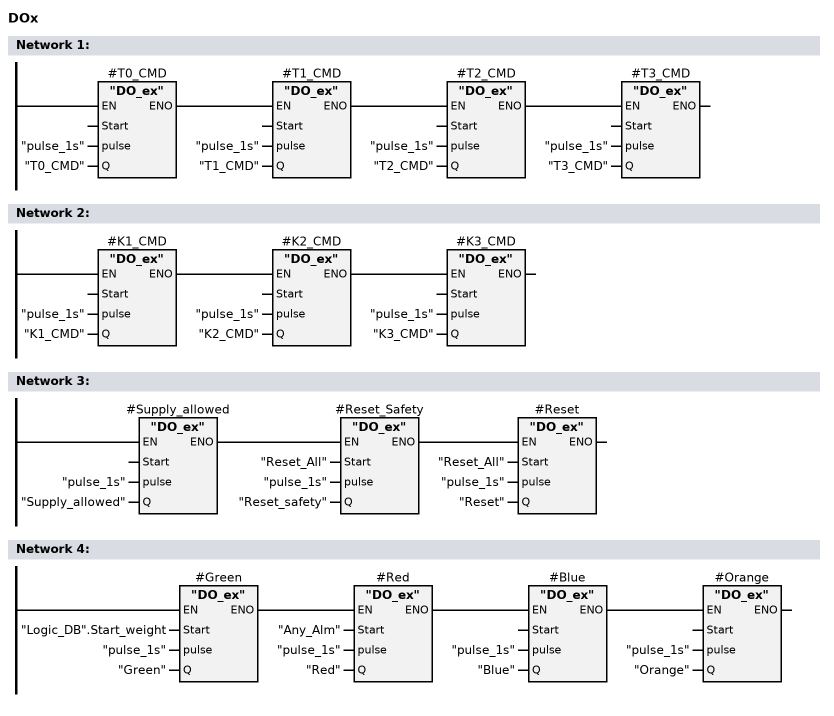
   RUNG wire#powerrail
      #T0_CMD(pulse := "pulse_1s", Q := "T0_CMD", Start :=)
      #T1_CMD(pulse := "pulse_1s", Q := "T1_CMD", Start :=)
      #T2_CMD(pulse := "pulse_1s", Q := "T2_CMD", Start :=)
      #T3_CMD(pulse := "pulse_1s", Q := "T3_CMD", Start :=)
   END_RUNG
   // the same network as SCL:
   #T0_CMD(pulse := "pulse_1s", Q := "T0_CMD", ENO => #_w1);   // "DO_ex"
   #T1_CMD(EN := #_w1, pulse := "pulse_1s", Q := "T1_CMD", ENO => #_w2);   // "DO_ex"
   #T2_CMD(EN := #_w2, pulse := "pulse_1s", Q := "T2_CMD", ENO => #_w3);   // "DO_ex"
   IF #_w3 THEN
       #T3_CMD(pulse := "pulse_1s", Q := "T3_CMD");   // "DO_ex"
   END_IF;
END_REGION

REGION Network 2
   RUNG wire#powerrail
      #K1_CMD(pulse := "pulse_1s", Q := "K1_CMD", Start :=)
      #K2_CMD(pulse := "pulse_1s", Q := "K2_CMD", Start :=)
      #K3_CMD(pulse := "pulse_1s", Q := "K3_CMD", Start :=)
   END_RUNG
   // the same network as SCL:
   #K1_CMD(pulse := "pulse_1s", Q := "K1_CMD", ENO => #_w1);   // "DO_ex"
   #K2_CMD(EN := #_w1, pulse := "pulse_1s", Q := "K2_CMD", ENO => #_w2);   // "DO_ex"
   IF #_w2 THEN
       #K3_CMD(pulse := "pulse_1s", Q := "K3_CMD");   // "DO_ex"
   END_IF;
END_REGION

REGION Network 3
   RUNG wire#powerrail
      #Supply_allowed(Start :=, pulse := "pulse_1s", Q := "Supply_allowed")
      #Reset_Safety(Start := "Reset_All", pulse := "pulse_1s", Q := "Reset_safety")
      #Reset(Start := "Reset_All", pulse := "pulse_1s", Q := "Reset")
   END_RUNG
   // the same network as SCL:
   #Supply_allowed(pulse := "pulse_1s", Q := "Supply_allowed", ENO => #_w1);   // "DO_ex"
   #Reset_Safety(EN := #_w1, Start := "Reset_All", pulse := "pulse_1s", Q := "Reset_safety", ENO => #_w2);   // "DO_ex"
   IF #_w2 THEN
       #Reset(Start := "Reset_All", pulse := "pulse_1s", Q := "Reset");   // "DO_ex"
   END_IF;
END_REGION

REGION Network 4
   RUNG wire#powerrail
      #Green(Start := "Logic_DB".Start_weight, pulse := "pulse_1s", Q := "Green")
      #Red(Start := "Any_Alm", pulse := "pulse_1s", Q := "Red")
      #Blue(Start :=, pulse := "pulse_1s", Q := "Blue")
      #Orange(Start :=, pulse := "pulse_1s", Q := "Orange")
   END_RUNG
   // the same network as SCL:
   #Green(Start := "Logic_DB".Start_weight, pulse := "pulse_1s", Q := "Green", ENO => #_w1);   // "DO_ex"
   #Red(EN := #_w1, Start := "Any_Alm", pulse := "pulse_1s", Q := "Red", ENO => #_w2);   // "DO_ex"
   #Blue(EN := #_w2, pulse := "pulse_1s", Q := "Blue", ENO => #_w3);   // "DO_ex"
   IF #_w3 THEN
       #Orange(pulse := "pulse_1s", Q := "Orange");   // "DO_ex"
   END_IF;
END_REGION
END_FUNCTION_BLOCK

// folder: System

FUNCTION_BLOCK "Tachometer"   // FB98, LAD
{ S7_Optimized_Access := 'FALSE' }
VERSION : 0.1
   VAR_INPUT
      Run : Bool;   // Управляющий сигнал
      Add : Bool;   // Один импульс
   END_VAR
   VAR_IN_OUT
      Result : Real;   // Текущая скорость, %
   END_VAR
   VAR
      Full : Real := 10.0;   // Кол-во импульсов на 1 оборот
      One : Real;   // Вес 1 импульса
      "A" : Real;   // Суммарный вес импульсов
      "B" : Real;   // Вес за последний цикл измерений
      T : Struct   // Уставка = времени одного оборота при 100% скорости
         SP : Real := 10.0;   // Уставка
         Now : Real;   // Текущий счёт
         One : Real;   // Вес импульса
         Progress : Real;   // Прогресс выполнения
         "Exit" : Bool;   // Счёт завершён
         Start : Bool;   // Запуск
         Pause : Bool;   // Пауза
         Reset : Bool;
         pos : Bool;   // Контроль фронта сигнала
      END_STRUCT;
   END_VAR
   VAR_TEMP
      pos_1 : Bool;
   END_VAR
   VAR_TEMP   // added for the SCL form of the ladder/FBD networks
      _w1 : Bool;
   END_VAR
BEGIN

REGION Network 1: Рассчёт веса импульса
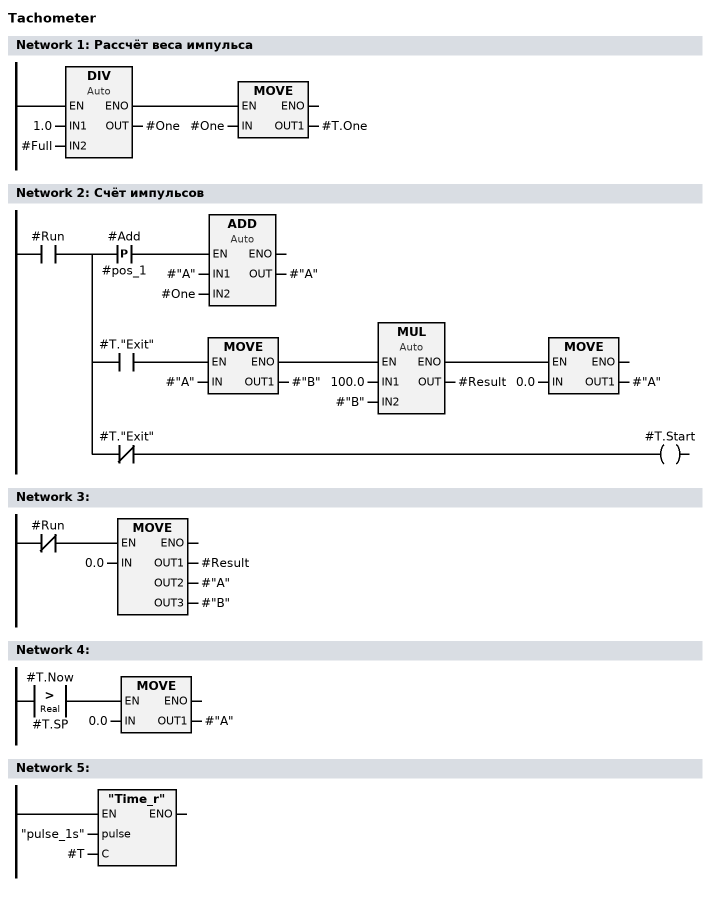
   RUNG wire#powerrail
      Div(in1 := 1.0, in2 := #Full, out => #One)
      Move(in := #One, out1 => #T.One)
   END_RUNG
   // the same network as SCL:
   #One := 1.0 / #Full;
   #T.One := #One;
END_REGION

REGION Network 2: Счёт импульсов
   RUNG wire#powerrail
      Contact( #Run )
      wire#w1
      P_Contact(operand := #Add, bit := #pos_1)
      Add(in1 := #"A", in2 := #One, out => #"A")
   END_RUNG
   RUNG wire#w1
      Contact( #T."Exit" )
      Move(in := #"A", out1 => #"B")
      Mul(in1 := 100.0, in2 := #"B", out => #Result)
      Move(in := 0.0, out1 => #"A")
   END_RUNG
   RUNG wire#w1
      I_Contact( #T."Exit" )
      Coil( #T.Start )
   END_RUNG
   // the same network as SCL:
   #_w1 := #Run AND #Add AND NOT #pos_1;   // rising edge of #Add
   #pos_1 := #Add;
   IF #_w1 THEN #"A" := #"A" + #One; END_IF;
   IF #Run AND #T."Exit" THEN
       #"B" := #"A";
       #Result := 100.0 * #"B";
       #"A" := 0.0;
   END_IF;
   #T.Start := #Run AND NOT #T."Exit";
END_REGION

REGION Network 3
   RUNG wire#powerrail
      I_Contact( #Run )
      Move(in := 0.0, out1 => #Result, out2 => #"A", out3 => #"B")
   END_RUNG
   // the same network as SCL:
   IF NOT #Run THEN
       #Result := 0.0;
       #"A" := 0.0;
       #"B" := 0.0;
   END_IF;
END_REGION

REGION Network 4
   RUNG wire#powerrail
      { S7_Templates := "SrcType := Real" } GT_Contact(in1 := #T.Now, in2 := #T.SP)
      Move(in := 0.0, out1 => #"A")
   END_RUNG
   // the same network as SCL:
   IF #T.Now > #T.SP THEN #"A" := 0.0; END_IF;
END_REGION

REGION Network 5
   RUNG wire#powerrail
      "Time_r"(pulse := "pulse_1s", C := #T)
   END_RUNG
   // the same network as SCL:
   "Time_r"(pulse := "pulse_1s", C := #T);
END_REGION
END_FUNCTION_BLOCK

FUNCTION_BLOCK "PID_ex"   // FB99, LAD
{ S7_Optimized_Access := 'FALSE' }
VERSION : 0.1
   VAR_INPUT
      Start : Bool;   // Команда запуска
      SP : Real;   // Уставка
      Value : Real;   // Показания датчика
   END_VAR
   VAR_IN_OUT
      Result : Real;   // Управляющее воздействие
   END_VAR
   VAR
      Hand : Bool;   // Ручной режим
      Err_Ack : Bool;   // Подтверждение аварии
      Reset : Bool;   // Сброс ПИД
      Error : Bool;   // Авария ПИД
      Invert : Bool;   // Инверсия работы
      SP_H : Bool;   // Авария уставки - превышение
      SP_L : Bool;   // Авария уставки - занижение
      In_H : Bool;   // Авария датчика - превышение
      In_L : Bool;   // Авария датчика - занижение
      Activate : Bool;   // Активировать ПИД
      Error_code : DWord;   // Код аварии
      Warning_code : DWord;   // Код предупреждения
      HandValue : Real;   // Выход ПИД в ручном режиме
      SP_P : Real := 1.5;   // Коэффициент пропорциональности
      SP_Ti : Real := 150.0;   // Время интегрирования
      SP_Td : Real;   // Время дифференцирования
      SP_Cycle : Real := 0.2;   // Время цикла
      Disturvance : Real;   // Внешнее воздействие
      Max_SP : Real := 500.0;   // Максимальное значение уставки
      Min_SP : Real := -500.0;   // Минимальное значение уставки
      Max_in : Real := 500.0;   // Максимальное значение датчика
      Min_in : Real := -500.0;   // Минимальное значение датчика
      Max_out : Real := 100.0;   // Максимальное значение выхода
      Min_out : Real := 0.0;   // Минимальное значение выхода
      "Type" : Int := 1;   // Режим работы
      State : Int;   // Состояние
      Mode : Int := 3;   // Режим
      PID : PID_Compact;   // ПИД
      DeadBand : Real;   // Мёртвая зона
      Max : Real;   // Верняя граница мёртвой зоны
      Min : Real;   // Нижняя граница мёртвой зоны
      Converter : Struct
         Use_Min_In : Bool;   // Отсекать входные значения ниже минимума
         Use_Max_In : Bool;   // Отсекать входные значения выше максимума
         Use_Min_Out : Bool;   // Отсекать результат ниже минимума
         Use_Max_Out : Bool;   // Отсекать результат выше максимума
         IO : Bool;   // Входной/Выходной режим
         Inverse : Bool;   // Инверсия выхода
         Min_In : Real := 0.0;   // Минимальный входной сигнал
         Max_In : Real := 100.0;   // Максимальный входной сигнал
         Min_Out : Real;   // Минимальный выходной сигнал
         Max_Out : Real;   // Максимальный выходной сигнал
      END_STRUCT;
      Conveter_Back : Struct
         Use_Min_In : Bool;   // Отсекать входные значения ниже минимума
         Use_Max_In : Bool;   // Отсекать входные значения выше максимума
         Use_Min_Out : Bool;   // Отсекать результат ниже минимума
         Use_Max_Out : Bool;   // Отсекать результат выше максимума
         IO : Bool;   // Входной/Выходной режим
         Inverse : Bool;   // Инверсия выхода
         Min_In : Real;   // Минимальный входной сигнал
         Max_In : Real;   // Максимальный входной сигнал
         Min_Out : Real := 0.0;   // Минимальный выходной сигнал
         Max_Out : Real := 100.0;   // Максимальный выходной сигнал
      END_STRUCT;
      C : Struct
         SP : Real := 1.0;   // Уставка
         Now : Real;   // Текущий счёт
         One : Real;   // Вес импульса
         Progress : Real;   // Прогресс выполнения
         "Exit" : Bool;   // Счёт завершён
         Start : Bool;   // Запуск
         Pause : Bool;   // Пауза
         Reset : Bool;   // Сброс счёта
         pos : Bool;   // Контроль фронта сигнала
      END_STRUCT;
   END_VAR
   VAR_TEMP
      PID_Output : Real;
   END_VAR
   VAR_TEMP   // added for the SCL form of the ladder/FBD networks
      _w1 : Bool;
   END_VAR
BEGIN

REGION Network 1: Сброс ПИД
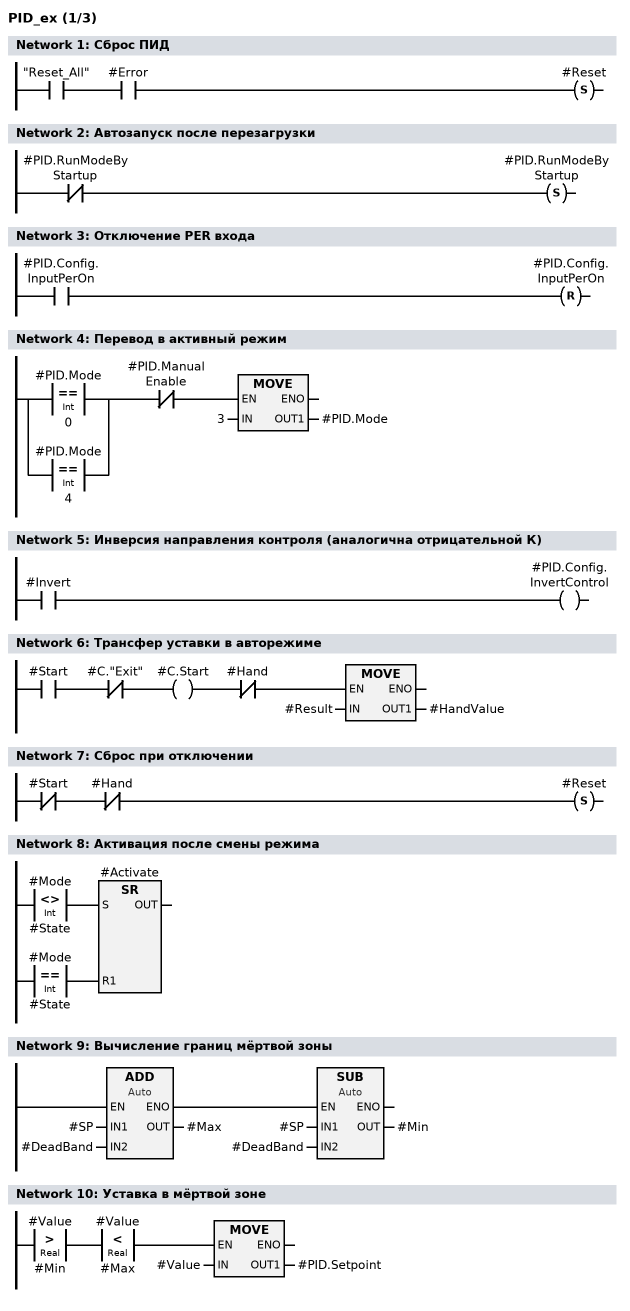
   RUNG wire#powerrail
      Contact( "Reset_All" )
      Contact( #Error )
      S_Coil( #Reset )
   END_RUNG
   // the same network as SCL:
   IF "Reset_All" AND #Error THEN #Reset := TRUE; END_IF;
END_REGION

REGION Network 2: Автозапуск после перезагрузки
   RUNG wire#powerrail
      I_Contact( #PID.RunModeByStartup )
      S_Coil( #PID.RunModeByStartup )
   END_RUNG
   // the same network as SCL:
   IF NOT #PID.RunModeByStartup THEN #PID.RunModeByStartup := TRUE; END_IF;
END_REGION

REGION Network 3: Отключение PER входа
   RUNG wire#powerrail
      Contact( #PID.Config.InputPerOn )
      R_Coil( #PID.Config.InputPerOn )
   END_RUNG
   // the same network as SCL:
   IF #PID.Config.InputPerOn THEN #PID.Config.InputPerOn := FALSE; END_IF;
END_REGION

REGION Network 4: Перевод в активный режим
   RUNG wire#powerrail
      { S7_Templates := "SrcType := Int" } EQ_Contact(in1 := #PID.Mode, in2 := 0)
      wire#w1
      I_Contact( #PID.ManualEnable )
      { S7_GenerateENO := "TRUE" } Move(in := 3, out1 => #PID.Mode)
   END_RUNG
   RUNG wire#powerrail
      { S7_Templates := "SrcType := Int" } EQ_Contact(in1 := #PID.Mode, in2 := 4)
   END_RUNG wire#w1
   // the same network as SCL:
   IF ((#PID.Mode = 0) OR (#PID.Mode = 4)) AND NOT #PID.ManualEnable THEN #PID.Mode := 3; END_IF;
END_REGION

REGION Network 5: Инверсия направления контроля (аналогична отрицательной К)
   RUNG wire#powerrail
      Contact( #Invert )
      Coil( #PID.Config.InvertControl )
   END_RUNG
   // the same network as SCL:
   #PID.Config.InvertControl := #Invert;
END_REGION

REGION Network 6: Трансфер уставки в авторежиме
   RUNG wire#powerrail
      Contact( #Start )
      I_Contact( #C."Exit" )
      Coil( #C.Start )
      I_Contact( #Hand )
      Move(in := #Result, out1 => #HandValue)
   END_RUNG
   // the same network as SCL:
   #C.Start := #Start AND NOT #C."Exit";
   IF #C.Start AND NOT #Hand THEN #HandValue := #Result; END_IF;
END_REGION

REGION Network 7: Сброс при отключении
   RUNG wire#powerrail
      I_Contact( #Start )
      I_Contact( #Hand )
      S_Coil( #Reset )
   END_RUNG
   // the same network as SCL:
   IF NOT #Start AND NOT #Hand THEN #Reset := TRUE; END_IF;
END_REGION

REGION Network 8: Активация после смены режима
   RUNG wire#powerrail
      { S7_Templates := "SrcType := Int" } NE_Contact(in1 := #Mode, in2 := #State)
      S_SR(operand := #Activate, r1 := wire#w1)
   END_RUNG
   RUNG wire#powerrail
      { S7_Templates := "SrcType := Int" } EQ_Contact(in1 := #Mode, in2 := #State)
   END_RUNG wire#w1
   // the same network as SCL:
   IF #Mode <> #State THEN
       #Activate := TRUE;   // SR flip-flop
   END_IF;
   IF #Mode = #State THEN #Activate := FALSE; END_IF;
END_REGION

REGION Network 9: Вычисление границ мёртвой зоны
   RUNG wire#powerrail
      Add(in1 := #SP, in2 := #DeadBand, out => #Max)
      Sub(in1 := #SP, in2 := #DeadBand, out => #Min)
   END_RUNG
   // the same network as SCL:
   #Max := #SP + #DeadBand;
   #Min := #SP - #DeadBand;
END_REGION

REGION Network 10: Уставка в мёртвой зоне
   RUNG wire#powerrail
      { S7_Templates := "SrcType := Real" } GT_Contact(in1 := #Value, in2 := #Min)
      { S7_Templates := "SrcType := Real" } LT_Contact(in1 := #Value, in2 := #Max)
      Move(in := #Value, out1 => #PID.Setpoint)
   END_RUNG
   // the same network as SCL:
   IF (#Value > #Min) AND (#Value < #Max) THEN #PID.Setpoint := #Value; END_IF;
END_REGION

REGION Network 11: Уставка вне мёртвой зоны
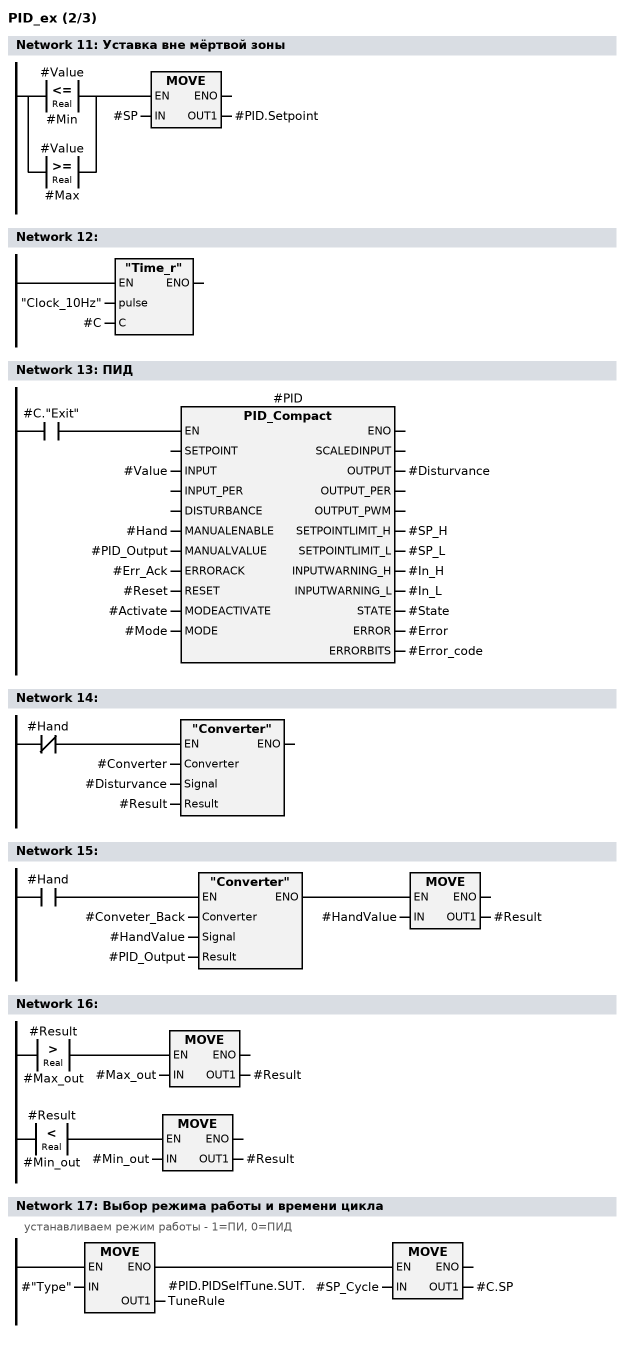
   RUNG wire#powerrail
      { S7_Templates := "SrcType := Real" } LE_Contact(in1 := #Value, in2 := #Min)
      wire#w1
      Move(in := #SP, out1 => #PID.Setpoint)
   END_RUNG
   RUNG wire#powerrail
      { S7_Templates := "SrcType := Real" } GE_Contact(in1 := #Value, in2 := #Max)
   END_RUNG wire#w1
   // the same network as SCL:
   IF (#Value <= #Min) OR (#Value >= #Max) THEN #PID.Setpoint := #SP; END_IF;
END_REGION

REGION Network 12
   RUNG wire#powerrail
      "Time_r"(pulse := "Clock_10Hz", C := #C)
   END_RUNG
   // the same network as SCL:
   "Time_r"(pulse := "Clock_10Hz", C := #C);
END_REGION

REGION Network 13: ПИД
   IF #C."Exit" THEN
       #PID(Input := #Value,   // PID_Compact
            ManualEnable := #Hand,
            ManualValue := #PID_Output,
            ErrorAck := #Err_Ack,
            Reset := #Reset,
            ModeActivate := #Activate,
            Mode := #Mode,
            Output => #Disturvance,
            SetpointLimit_H => #SP_H,
            SetpointLimit_L => #SP_L,
            InputWarning_H => #In_H,
            InputWarning_L => #In_L,
            State => #State,
            Error => #Error,
            ErrorBits => #Error_code);
   END_IF;
END_REGION

REGION Network 14
   RUNG wire#powerrail
      I_Contact( #Hand )
      "Converter"(Converter := #Converter, Signal := #Disturvance, Result := #Result)
   END_RUNG
   // the same network as SCL:
   IF NOT #Hand THEN "Converter"(Converter := #Converter, Signal := #Disturvance, Result := #Result); END_IF;
END_REGION

REGION Network 15
   RUNG wire#powerrail
      Contact( #Hand )
      "Converter"(Converter := #Conveter_Back, Signal := #HandValue, Result := #PID_Output)
      Move(in := #HandValue, out1 => #Result)
   END_RUNG
   // the same network as SCL:
   "Converter"(EN := #Hand,
               Converter := #Conveter_Back,
               Signal := #HandValue,
               Result := #PID_Output,
               ENO => #_w1);
   IF #_w1 THEN #Result := #HandValue; END_IF;
END_REGION

REGION Network 16
   RUNG wire#powerrail
      { S7_Templates := "SrcType := Real" } GT_Contact(in1 := #Result, in2 := #Max_out)
      Move(in := #Max_out, out1 => #Result)
   END_RUNG
   RUNG wire#powerrail
      { S7_Templates := "SrcType := Real" } LT_Contact(in1 := #Result, in2 := #Min_out)
      Move(in := #Min_out, out1 => #Result)
   END_RUNG
   // the same network as SCL:
   IF #Result > #Max_out THEN #Result := #Max_out; END_IF;
   IF #Result < #Min_out THEN #Result := #Min_out; END_IF;
END_REGION

REGION Network 17: Выбор режима работы и времени цикла
   // устанавливаем режим работы - 1=ПИ, 0=ПИД
   RUNG wire#powerrail
      { S7_GenerateENO := "TRUE" } Move(in := #"Type", out1 => #PID.PIDSelfTune.SUT.TuneRule)
      { S7_GenerateENO := "TRUE" } Move(in := #SP_Cycle, out1 => #C.SP)
   END_RUNG
   // the same network as SCL:
   // ENO of a box is taken as its EN; it also drops when the box reports an error
   #PID.PIDSelfTune.SUT.TuneRule := #"Type";
   #C.SP := #SP_Cycle;
END_REGION

REGION Network 18: Параметры регулирования
   // Задаём коэффициент пропорциональности и время интегрирования.
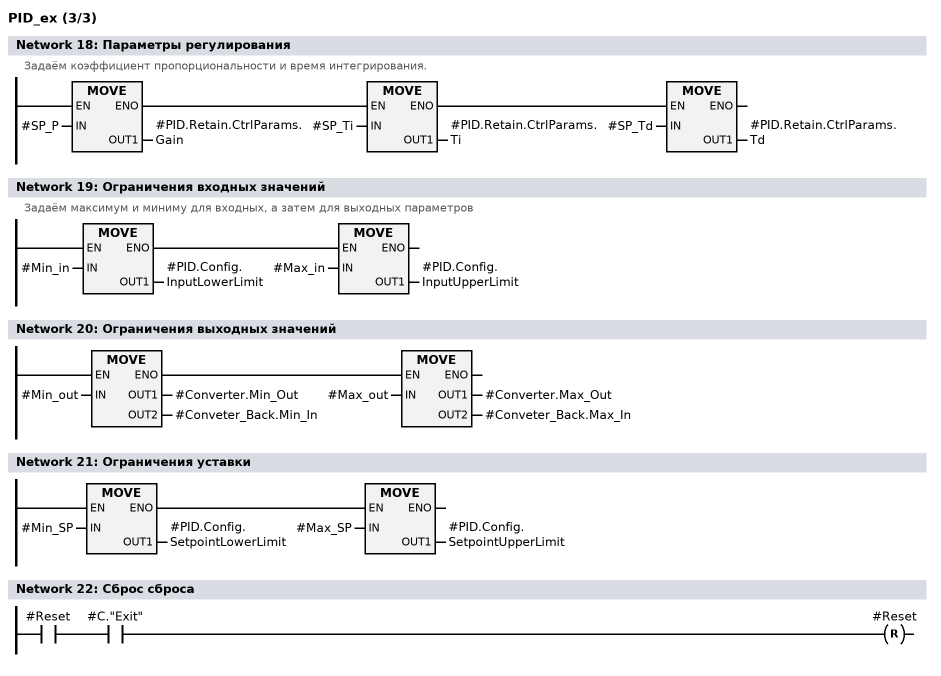
   RUNG wire#powerrail
      { S7_GenerateENO := "TRUE" } Move(in := #SP_P, out1 => #PID.Retain.CtrlParams.Gain)
      { S7_GenerateENO := "TRUE" } Move(in := #SP_Ti, out1 => #PID.Retain.CtrlParams.Ti)
      { S7_GenerateENO := "TRUE" } Move(in := #SP_Td, out1 => #PID.Retain.CtrlParams.Td)
   END_RUNG
   // the same network as SCL:
   // ENO of a box is taken as its EN; it also drops when the box reports an error
   #PID.Retain.CtrlParams.Gain := #SP_P;
   #PID.Retain.CtrlParams.Ti := #SP_Ti;
   #PID.Retain.CtrlParams.Td := #SP_Td;
END_REGION

REGION Network 19: Ограничения входных значений
   // Задаём максимум и миниму для входных, а затем для выходных параметров
   RUNG wire#powerrail
      { S7_GenerateENO := "TRUE" } Move(in := #Min_in, out1 => #PID.Config.InputLowerLimit)
      { S7_GenerateENO := "TRUE" } Move(in := #Max_in, out1 => #PID.Config.InputUpperLimit)
   END_RUNG
   // the same network as SCL:
   // ENO of a box is taken as its EN; it also drops when the box reports an error
   #PID.Config.InputLowerLimit := #Min_in;
   #PID.Config.InputUpperLimit := #Max_in;
END_REGION

REGION Network 20: Ограничения выходных значений
   RUNG wire#powerrail
      { S7_GenerateENO := "TRUE" } Move(in := #Min_out, out1 => #Converter.Min_Out, out2 => #Conveter_Back.Min_In)
      { S7_GenerateENO := "TRUE" } Move(in := #Max_out, out1 => #Converter.Max_Out, out2 => #Conveter_Back.Max_In)
   END_RUNG
   // the same network as SCL:
   // ENO of a box is taken as its EN; it also drops when the box reports an error
   #Converter.Min_Out := #Min_out;
   #Conveter_Back.Min_In := #Min_out;
   #Converter.Max_Out := #Max_out;
   #Conveter_Back.Max_In := #Max_out;
END_REGION

REGION Network 21: Ограничения уставки
   RUNG wire#powerrail
      { S7_GenerateENO := "TRUE" } Move(in := #Min_SP, out1 => #PID.Config.SetpointLowerLimit)
      { S7_GenerateENO := "TRUE" } Move(in := #Max_SP, out1 => #PID.Config.SetpointUpperLimit)
   END_RUNG
   // the same network as SCL:
   // ENO of a box is taken as its EN; it also drops when the box reports an error
   #PID.Config.SetpointLowerLimit := #Min_SP;
   #PID.Config.SetpointUpperLimit := #Max_SP;
END_REGION

REGION Network 22: Сброс сброса
   RUNG wire#powerrail
      Contact( #Reset )
      Contact( #C."Exit" )
      R_Coil( #Reset )
   END_RUNG
   // the same network as SCL:
   IF #Reset AND #C."Exit" THEN #Reset := FALSE; END_IF;
END_REGION
END_FUNCTION_BLOCK

FUNCTION "DRV_pulse" : Void   // FC100, LAD
{ S7_Optimized_Access := 'FALSE' }
VERSION : 0.1
   VAR_TEMP   // added for the SCL form of the ladder/FBD networks
      _w1 : Bool;
      _w2 : Bool;
   END_VAR
BEGIN

REGION Network 1
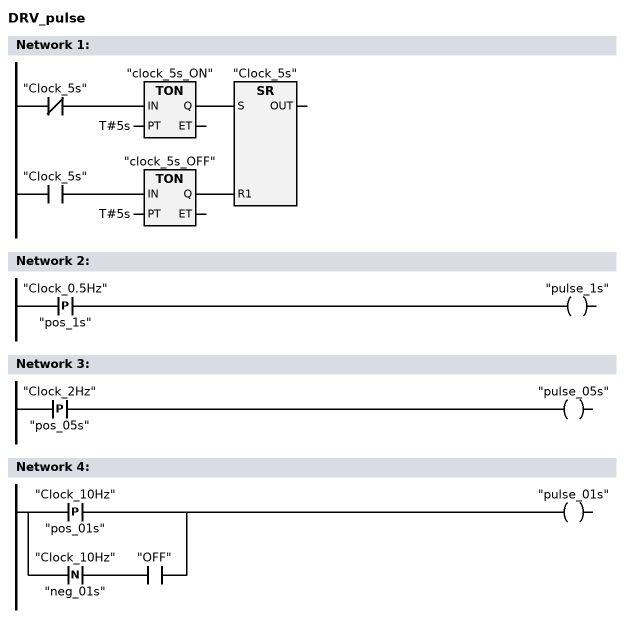
   "clock_5s_ON".TON(IN := NOT "Clock_5s", PT := T#5s);
   "clock_5s_OFF".TON(IN := "Clock_5s", PT := T#5s);
   IF "clock_5s_ON".Q THEN
       "Clock_5s" := TRUE;   // SR flip-flop
   END_IF;
   IF "clock_5s_OFF".Q THEN "Clock_5s" := FALSE; END_IF;
END_REGION

REGION Network 2
   RUNG wire#powerrail
      P_Contact(operand := "Clock_0.5Hz", bit := "pos_1s")
      Coil( "pulse_1s" )
   END_RUNG
   // the same network as SCL:
   #_w1 := "Clock_0.5Hz" AND NOT "pos_1s";   // rising edge of "Clock_0.5Hz"
   "pos_1s" := "Clock_0.5Hz";
   "pulse_1s" := #_w1;
END_REGION

REGION Network 3
   RUNG wire#powerrail
      P_Contact(operand := "Clock_2Hz", bit := "pos_05s")
      Coil( "pulse_05s" )
   END_RUNG
   // the same network as SCL:
   #_w1 := "Clock_2Hz" AND NOT "pos_05s";   // rising edge of "Clock_2Hz"
   "pos_05s" := "Clock_2Hz";
   "pulse_05s" := #_w1;
END_REGION

REGION Network 4
   RUNG wire#powerrail
      P_Contact(operand := "Clock_10Hz", bit := "pos_01s")
      wire#w1
      Coil( "pulse_01s" )
   END_RUNG
   RUNG wire#powerrail
      N_Contact(operand := "Clock_10Hz", bit := "neg_01s")
      Contact( "OFF" )
   END_RUNG wire#w1
   // the same network as SCL:
   #_w1 := "Clock_10Hz" AND NOT "pos_01s";   // rising edge of "Clock_10Hz"
   "pos_01s" := "Clock_10Hz";
   #_w2 := NOT "Clock_10Hz" AND "neg_01s";   // falling edge of "Clock_10Hz"
   "neg_01s" := "Clock_10Hz";
   "pulse_01s" := #_w1 OR (#_w2 AND "OFF");
END_REGION
END_FUNCTION

FUNCTION "DRV_End" : Void   // FC101, LAD
{ S7_Optimized_Access := 'TRUE' }
VERSION : 0.1
BEGIN

REGION Network 1: Одно из устройств нижнего уровня в ручном режиме
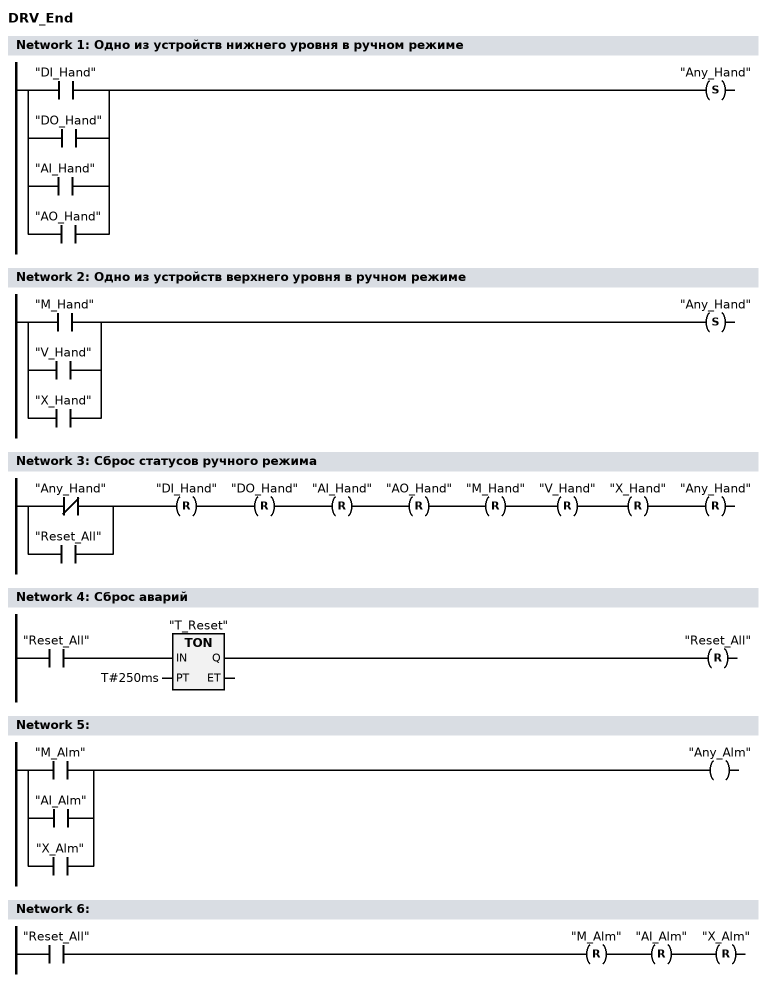
   RUNG wire#powerrail
      Contact( "DI_Hand" )
      wire#w1
      S_Coil( "Any_Hand" )
   END_RUNG
   RUNG wire#powerrail
      Contact( "DO_Hand" )
   END_RUNG wire#w1
   RUNG wire#powerrail
      Contact( "AI_Hand" )
   END_RUNG wire#w1
   RUNG wire#powerrail
      Contact( "AO_Hand" )
   END_RUNG wire#w1
   // the same network as SCL:
   IF "DI_Hand" OR "DO_Hand" OR "AI_Hand" OR "AO_Hand" THEN "Any_Hand" := TRUE; END_IF;
END_REGION

REGION Network 2: Одно из устройств верхнего уровня в ручном режиме
   RUNG wire#powerrail
      Contact( "M_Hand" )
      wire#w1
      S_Coil( "Any_Hand" )
   END_RUNG
   RUNG wire#powerrail
      Contact( "V_Hand" )
   END_RUNG wire#w1
   RUNG wire#powerrail
      Contact( "X_Hand" )
   END_RUNG wire#w1
   // the same network as SCL:
   IF "M_Hand" OR "V_Hand" OR "X_Hand" THEN "Any_Hand" := TRUE; END_IF;
END_REGION

REGION Network 3: Сброс статусов ручного режима
   RUNG wire#powerrail
      I_Contact( "Any_Hand" )
      wire#w1
      R_Coil( "DI_Hand" )
      R_Coil( "DO_Hand" )
      R_Coil( "AI_Hand" )
      R_Coil( "AO_Hand" )
      R_Coil( "M_Hand" )
      R_Coil( "V_Hand" )
      R_Coil( "X_Hand" )
      R_Coil( "Any_Hand" )
   END_RUNG
   RUNG wire#powerrail
      Contact( "Reset_All" )
   END_RUNG wire#w1
   // the same network as SCL:
   IF NOT "Any_Hand" OR "Reset_All" THEN
       "DI_Hand" := FALSE;
       "DO_Hand" := FALSE;
       "AI_Hand" := FALSE;
       "AO_Hand" := FALSE;
       "M_Hand" := FALSE;
       "V_Hand" := FALSE;
       "X_Hand" := FALSE;
       "Any_Hand" := FALSE;
   END_IF;
END_REGION

REGION Network 4: Сброс аварий
   "T_Reset".TON(IN := "Reset_All", PT := T#250ms);
   IF "T_Reset".Q THEN "Reset_All" := FALSE; END_IF;
END_REGION

REGION Network 5
   RUNG wire#powerrail
      Contact( "M_Alm" )
      wire#w1
      Coil( "Any_Alm" )
   END_RUNG
   RUNG wire#powerrail
      Contact( "AI_Alm" )
   END_RUNG wire#w1
   RUNG wire#powerrail
      Contact( "X_Alm" )
   END_RUNG wire#w1
   // the same network as SCL:
   "Any_Alm" := "M_Alm" OR "AI_Alm" OR "X_Alm";
END_REGION

REGION Network 6
   RUNG wire#powerrail
      Contact( "Reset_All" )
      R_Coil( "M_Alm" )
      R_Coil( "AI_Alm" )
      R_Coil( "X_Alm" )
   END_RUNG
   // the same network as SCL:
   IF "Reset_All" THEN
       "M_Alm" := FALSE;
       "AI_Alm" := FALSE;
       "X_Alm" := FALSE;
   END_IF;
END_REGION
END_FUNCTION

FUNCTION "Converter" : Void   // FC102, LAD
TITLE = Драйвер линеаризации аналогового сигнала
{ S7_Optimized_Access := 'FALSE' }
VERSION : 0.1
   VAR_INPUT
      Converter : Struct
         Use_Min_In : Bool;   // Отсекать входные значения ниже минимума
         Use_Max_In : Bool;   // Отсекать входные значения выше максимума
         Use_Min_Out : Bool;   // Отсекать результат ниже минимума
         Use_Max_Out : Bool;   // Отсекать результат выше максимума
         IO : Bool;   // Входной/Выходной режим
         Inverse : Bool;   // Инверсия выхода
         Min_In : Real;   // Минимальный входной сигнал
         Max_In : Real;   // Максимальный входной сигнал
         Min_Out : Real;   // Минимальный выходной сигнал
         Max_Out : Real;   // Максимальный выходной сигнал
      END_STRUCT;
   END_VAR
   VAR_IN_OUT
      Signal : Real;   // Входной сигнал
      Result : Real;   // Результат линеаризации
   END_VAR
   VAR_TEMP
      Range_In : Real;   // Диапазон входного сигнала
      Range_Out : Real;   // Диапазон выходного сигнала
      T_T : Real;   // Соотношение диапазонов
      R_Sig : Real;   // Поправка на отрицательные значения
   END_VAR
BEGIN

REGION Network 1: Проверка нижнего уровня входного сигнала
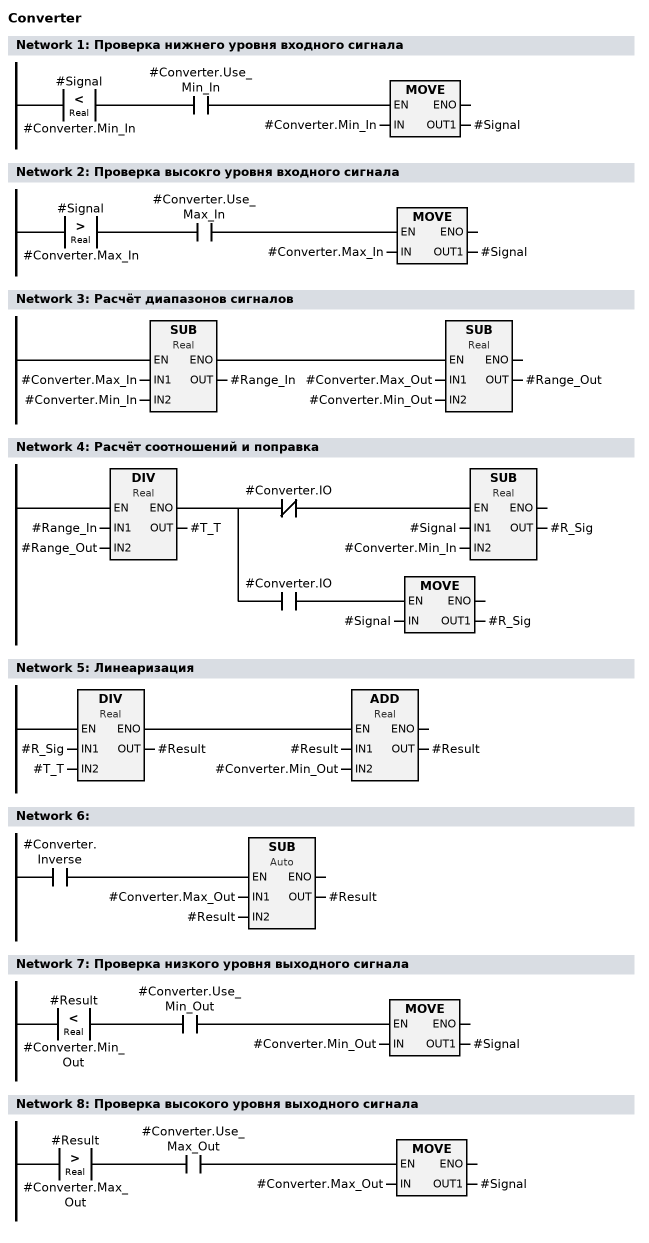
   RUNG wire#powerrail
      { S7_Templates := "SrcType := Real" } LT_Contact(in1 := #Signal, in2 := #Converter.Min_In)
      Contact( #Converter.Use_Min_In )
      Move(in := #Converter.Min_In, out1 => #Signal)
   END_RUNG
   // the same network as SCL:
   IF (#Signal < #Converter.Min_In) AND #Converter.Use_Min_In THEN #Signal := #Converter.Min_In; END_IF;
END_REGION

REGION Network 2: Проверка высокго уровня входного сигнала
   RUNG wire#powerrail
      { S7_Templates := "SrcType := Real" } GT_Contact(in1 := #Signal, in2 := #Converter.Max_In)
      Contact( #Converter.Use_Max_In )
      Move(in := #Converter.Max_In, out1 => #Signal)
   END_RUNG
   // the same network as SCL:
   IF (#Signal > #Converter.Max_In) AND #Converter.Use_Max_In THEN #Signal := #Converter.Max_In; END_IF;
END_REGION

REGION Network 3: Расчёт диапазонов сигналов
   RUNG wire#powerrail
      { S7_Templates := "SrcType := Real"; S7_GenerateENO := "TRUE" } Sub(in1 := #Converter.Max_In, in2 := #Converter.Min_In, out => #Range_In)
      { S7_Templates := "SrcType := Real"; S7_GenerateENO := "TRUE" } Sub(in1 := #Converter.Max_Out, in2 := #Converter.Min_Out, out => #Range_Out)
   END_RUNG
   // the same network as SCL:
   // ENO of a box is taken as its EN; it also drops when the box reports an error
   #Range_In := #Converter.Max_In - #Converter.Min_In;
   #Range_Out := #Converter.Max_Out - #Converter.Min_Out;
END_REGION

REGION Network 4: Расчёт соотношений и поправка
   RUNG wire#powerrail
      { S7_Templates := "SrcType := Real"; S7_GenerateENO := "TRUE" } Div(in1 := #Range_In, in2 := #Range_Out, out => #T_T)
      wire#w1
      I_Contact( #Converter.IO )
      { S7_Templates := "SrcType := Real"; S7_GenerateENO := "TRUE" } Sub(in1 := #Signal, in2 := #Converter.Min_In, out => #R_Sig)
   END_RUNG
   RUNG wire#w1
      Contact( #Converter.IO )
      Move(in := #Signal, out1 => #R_Sig)
   END_RUNG
   // the same network as SCL:
   // ENO of a box is taken as its EN; it also drops when the box reports an error
   #T_T := #Range_In / #Range_Out;
   IF NOT #Converter.IO THEN #R_Sig := #Signal - #Converter.Min_In; END_IF;
   IF #Converter.IO THEN #R_Sig := #Signal; END_IF;
END_REGION

REGION Network 5: Линеаризация
   RUNG wire#powerrail
      { S7_Templates := "SrcType := Real"; S7_GenerateENO := "TRUE" } Div(in1 := #R_Sig, in2 := #T_T, out => #Result)
      { S7_Templates := "SrcType := Real"; S7_GenerateENO := "TRUE" } Add(in1 := #Result, in2 := #Converter.Min_Out, out => #Result)
   END_RUNG
   // the same network as SCL:
   // ENO of a box is taken as its EN; it also drops when the box reports an error
   #Result := #R_Sig / #T_T;
   #Result := #Result + #Converter.Min_Out;
END_REGION

REGION Network 6
   RUNG wire#powerrail
      Contact( #Converter.Inverse )
      Sub(in1 := #Converter.Max_Out, in2 := #Result, out => #Result)
   END_RUNG
   // the same network as SCL:
   IF #Converter.Inverse THEN #Result := #Converter.Max_Out - #Result; END_IF;
END_REGION

REGION Network 7: Проверка низкого уровня выходного сигнала
   RUNG wire#powerrail
      { S7_Templates := "SrcType := Real" } LT_Contact(in1 := #Result, in2 := #Converter.Min_Out)
      Contact( #Converter.Use_Min_Out )
      Move(in := #Converter.Min_Out, out1 => #Signal)
   END_RUNG
   // the same network as SCL:
   IF (#Result < #Converter.Min_Out) AND #Converter.Use_Min_Out THEN #Signal := #Converter.Min_Out; END_IF;
END_REGION

REGION Network 8: Проверка высокого уровня выходного сигнала
   RUNG wire#powerrail
      { S7_Templates := "SrcType := Real" } GT_Contact(in1 := #Result, in2 := #Converter.Max_Out)
      Contact( #Converter.Use_Max_Out )
      Move(in := #Converter.Max_Out, out1 => #Signal)
   END_RUNG
   // the same network as SCL:
   IF (#Result > #Converter.Max_Out) AND #Converter.Use_Max_Out THEN #Signal := #Converter.Max_Out; END_IF;
END_REGION
END_FUNCTION

FUNCTION "Balancer" : Void   // FC103, LAD
TITLE = Балансировка нагрузки двух устройств по наработке и аварии
{ S7_Optimized_Access := 'FALSE' }
VERSION : 0.1
   VAR_INPUT
      CMD : Bool;   // Команда запуска
      Res_1 : DInt;   // Наработка устройства 1
      Res_2 : DInt;   // Наработка устройства 2
      Alm_1 : Bool;   // Авария устройства 1
      Alm_2 : Bool;   // Авария устройства 2
   END_VAR
   VAR_IN_OUT
      Res_SP : DInt;   // Переключение по наработке
      CMD_1 : Bool;   // Команда на устройство 1
      CMD_2 : Bool;   // Команда на устройство 2
   END_VAR
   VAR_TEMP
      N : Bool;   // Выбор устройства
      Now : DInt;   // Текущая разница наработок
   END_VAR
BEGIN

REGION Network 1: Подсчёт разницы наработки
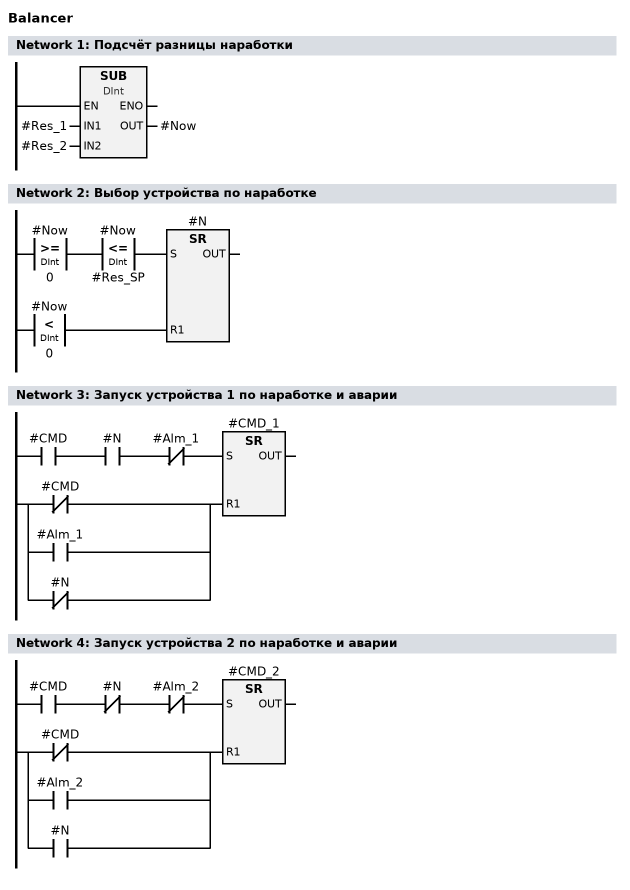
   RUNG wire#powerrail
      { S7_Templates := "SrcType := DInt"; S7_GenerateENO := "TRUE" } Sub(in1 := #Res_1, in2 := #Res_2, out => #Now)
   END_RUNG
   // the same network as SCL:
   #Now := #Res_1 - #Res_2;
END_REGION

REGION Network 2: Выбор устройства по наработке
   RUNG wire#powerrail
      { S7_Templates := "SrcType := DInt" } GE_Contact(in1 := #Now, in2 := 0)
      { S7_Templates := "SrcType := DInt" } LE_Contact(in1 := #Now, in2 := #Res_SP)
      S_SR(operand := #N, r1 := wire#w1)
   END_RUNG
   RUNG wire#powerrail
      { S7_Templates := "SrcType := DInt" } LT_Contact(in1 := #Now, in2 := 0)
   END_RUNG wire#w1
   // the same network as SCL:
   IF (#Now >= 0) AND (#Now <= #Res_SP) THEN
       #N := TRUE;   // SR flip-flop
   END_IF;
   IF #Now < 0 THEN #N := FALSE; END_IF;
END_REGION

REGION Network 3: Запуск устройства 1 по наработке и аварии
   RUNG wire#powerrail
      Contact( #CMD )
      Contact( #N )
      I_Contact( #Alm_1 )
      S_SR(operand := #CMD_1, r1 := wire#w1)
   END_RUNG
   RUNG wire#powerrail
      I_Contact( #CMD )
   END_RUNG wire#w1
   RUNG wire#powerrail
      Contact( #Alm_1 )
   END_RUNG wire#w1
   RUNG wire#powerrail
      I_Contact( #N )
   END_RUNG wire#w1
   // the same network as SCL:
   IF #CMD AND #N AND NOT #Alm_1 THEN
       #CMD_1 := TRUE;   // SR flip-flop
   END_IF;
   IF NOT #CMD OR #Alm_1 OR NOT #N THEN #CMD_1 := FALSE; END_IF;
END_REGION

REGION Network 4: Запуск устройства 2 по наработке и аварии
   RUNG wire#powerrail
      Contact( #CMD )
      I_Contact( #N )
      I_Contact( #Alm_2 )
      S_SR(operand := #CMD_2, r1 := wire#w1)
   END_RUNG
   RUNG wire#powerrail
      I_Contact( #CMD )
   END_RUNG wire#w1
   RUNG wire#powerrail
      Contact( #Alm_2 )
   END_RUNG wire#w1
   RUNG wire#powerrail
      Contact( #N )
   END_RUNG wire#w1
   // the same network as SCL:
   IF #CMD AND NOT #N AND NOT #Alm_2 THEN
       #CMD_2 := TRUE;   // SR flip-flop
   END_IF;
   IF NOT #CMD OR #Alm_2 OR #N THEN #CMD_2 := FALSE; END_IF;
END_REGION
END_FUNCTION

FUNCTION "Time_s" : Void   // FC104, LAD
{ S7_Optimized_Access := 'FALSE' }
VERSION : 0.1
   VAR_INPUT
      pulse : Bool;
   END_VAR
   VAR_IN_OUT
      T : Struct
         SP : Int;   // Уставка
         Now : Int;   // Текущий счёт
         "Exit" : Bool;   // Счёт завершён
         Start : Bool;   // Запуск
         Pause : Bool;   // Пауза
         Reset : Bool;   // Сброс таймера
      END_STRUCT;
   END_VAR
   VAR_TEMP   // added for the SCL form of the ladder/FBD networks
      _w1 : Bool;
   END_VAR
BEGIN

REGION Network 1: Подсчёт времени
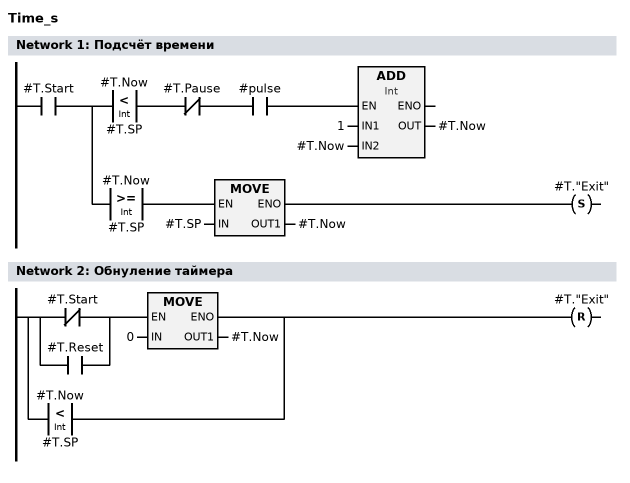
   RUNG wire#powerrail
      Contact( #T.Start )
      wire#w1
      { S7_Templates := "SrcType := Int" } LT_Contact(in1 := #T.Now, in2 := #T.SP)
      I_Contact( #T.Pause )
      Contact( #pulse )
      { S7_Templates := "SrcType := Int"; S7_GenerateENO := "TRUE" } Add(in1 := 1, in2 := #T.Now, out => #T.Now)
   END_RUNG
   RUNG wire#w1
      { S7_Templates := "SrcType := Int" } GE_Contact(in1 := #T.Now, in2 := #T.SP)
      Move(in := #T.SP, out1 => #T.Now)
      S_Coil( #T."Exit" )
   END_RUNG
   // the same network as SCL:
   IF #T.Start AND (#T.Now < #T.SP) AND NOT #T.Pause AND #pulse THEN #T.Now := 1 + #T.Now; END_IF;
   #_w1 := #T.Start AND (#T.Now >= #T.SP);
   IF #_w1 THEN
       #T.Now := #T.SP;
       #T."Exit" := TRUE;
   END_IF;
END_REGION

REGION Network 2: Обнуление таймера
   RUNG wire#powerrail
      I_Contact( #T.Start )
      wire#w1
      { S7_GenerateENO := "TRUE" } Move(in := 0, out1 => #T.Now)
      wire#w2
      R_Coil( #T."Exit" )
   END_RUNG
   RUNG wire#powerrail
      Contact( #T.Reset )
   END_RUNG wire#w1
   RUNG wire#powerrail
      { S7_Templates := "SrcType := Int" } LT_Contact(in1 := #T.Now, in2 := #T.SP)
   END_RUNG wire#w2
   // the same network as SCL:
   // ENO of a box is taken as its EN; it also drops when the box reports an error
   #_w1 := NOT #T.Start OR #T.Reset;
   IF #_w1 THEN #T.Now := 0; END_IF;
   IF #_w1 OR (#T.Now < #T.SP) THEN #T."Exit" := FALSE; END_IF;
END_REGION
END_FUNCTION

FUNCTION "Time_m" : Void   // FC105, LAD
{ S7_Optimized_Access := 'FALSE' }
VERSION : 0.1
   VAR_INPUT
      pulse : Bool;
   END_VAR
   VAR_IN_OUT
      T : Struct
         SP_M : Int;   // Уставка минут
         SP_S : Int;   // Уставка секунд
         Now_M : Int;   // Текущий счёт минут
         Now_S : Int;   // Текущий счёт секунд
         "Exit" : Bool;   // Счёт завершён
         Start : Bool;   // Запуск
         Pause : Bool;   // Пауза
         Reset : Bool;   // Сброс таймера
      END_STRUCT;
   END_VAR
   VAR_TEMP   // added for the SCL form of the ladder/FBD networks
      _w1 : Bool;
   END_VAR
BEGIN

REGION Network 1: Подсчёт времени
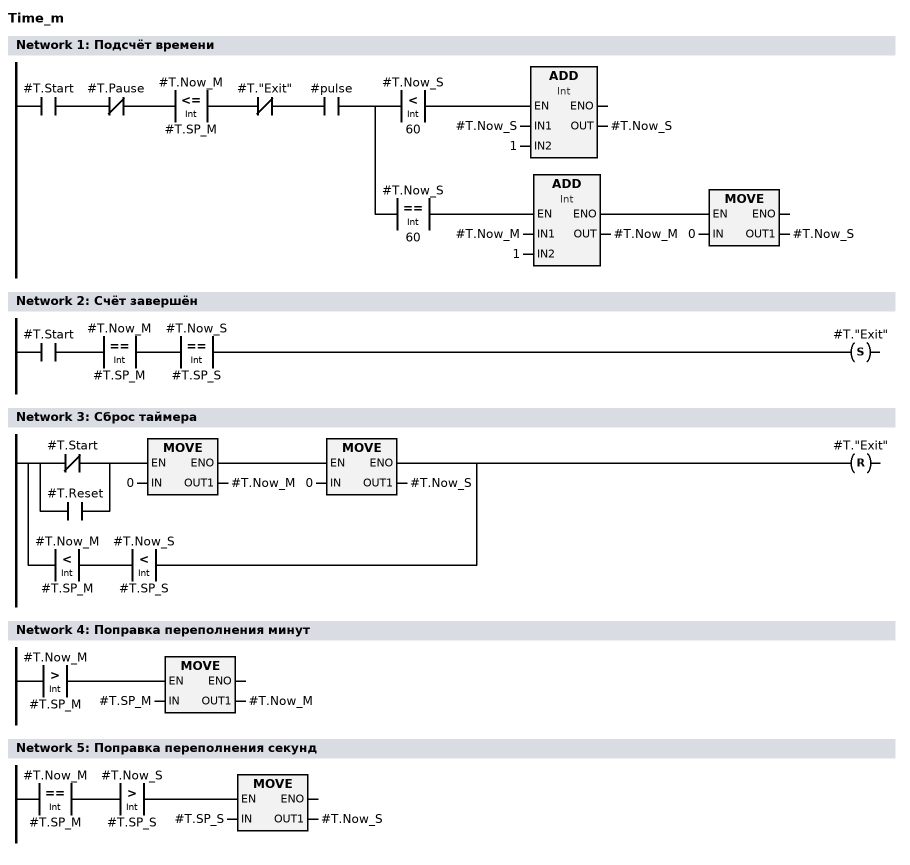
   RUNG wire#powerrail
      Contact( #T.Start )
      I_Contact( #T.Pause )
      { S7_Templates := "SrcType := Int" } LE_Contact(in1 := #T.Now_M, in2 := #T.SP_M)
      I_Contact( #T."Exit" )
      Contact( #pulse )
      wire#w1
      { S7_Templates := "SrcType := Int" } LT_Contact(in1 := #T.Now_S, in2 := 60)
      { S7_Templates := "SrcType := Int"; S7_GenerateENO := "TRUE" } Add(in1 := #T.Now_S, in2 := 1, out => #T.Now_S)
   END_RUNG
   RUNG wire#w1
      { S7_Templates := "SrcType := Int" } EQ_Contact(in1 := #T.Now_S, in2 := 60)
      { S7_Templates := "SrcType := Int"; S7_GenerateENO := "TRUE" } Add(in1 := #T.Now_M, in2 := 1, out => #T.Now_M)
      Move(in := 0, out1 => #T.Now_S)
   END_RUNG
   // the same network as SCL:
   // ENO of a box is taken as its EN; it also drops when the box reports an error
   #_w1 := #T.Start AND NOT #T.Pause AND (#T.Now_M <= #T.SP_M) AND NOT #T."Exit" AND #pulse;
   IF #_w1 AND (#T.Now_S < 60) THEN #T.Now_S := #T.Now_S + 1; END_IF;
   IF #_w1 AND (#T.Now_S = 60) THEN
       #T.Now_M := #T.Now_M + 1;
       #T.Now_S := 0;
   END_IF;
END_REGION

REGION Network 2: Счёт завершён
   RUNG wire#powerrail
      Contact( #T.Start )
      { S7_Templates := "SrcType := Int" } EQ_Contact(in1 := #T.Now_M, in2 := #T.SP_M)
      { S7_Templates := "SrcType := Int" } EQ_Contact(in1 := #T.Now_S, in2 := #T.SP_S)
      S_Coil( #T."Exit" )
   END_RUNG
   // the same network as SCL:
   IF #T.Start AND (#T.Now_M = #T.SP_M) AND (#T.Now_S = #T.SP_S) THEN #T."Exit" := TRUE; END_IF;
END_REGION

REGION Network 3: Сброс таймера
   RUNG wire#powerrail
      I_Contact( #T.Start )
      wire#w1
      { S7_GenerateENO := "TRUE" } Move(in := 0, out1 => #T.Now_M)
      { S7_GenerateENO := "TRUE" } Move(in := 0, out1 => #T.Now_S)
      wire#w2
      R_Coil( #T."Exit" )
   END_RUNG
   RUNG wire#powerrail
      Contact( #T.Reset )
   END_RUNG wire#w1
   RUNG wire#powerrail
      { S7_Templates := "SrcType := Int" } LT_Contact(in1 := #T.Now_M, in2 := #T.SP_M)
      { S7_Templates := "SrcType := Int" } LT_Contact(in1 := #T.Now_S, in2 := #T.SP_S)
   END_RUNG wire#w2
   // the same network as SCL:
   // ENO of a box is taken as its EN; it also drops when the box reports an error
   #_w1 := NOT #T.Start OR #T.Reset;
   IF #_w1 THEN
       #T.Now_M := 0;
       #T.Now_S := 0;
   END_IF;
   IF #_w1 OR ((#T.Now_M < #T.SP_M) AND (#T.Now_S < #T.SP_S)) THEN #T."Exit" := FALSE; END_IF;
END_REGION

REGION Network 4: Поправка переполнения минут
   RUNG wire#powerrail
      { S7_Templates := "SrcType := Int" } GT_Contact(in1 := #T.Now_M, in2 := #T.SP_M)
      { S7_GenerateENO := "TRUE" } Move(in := #T.SP_M, out1 => #T.Now_M)
   END_RUNG
   // the same network as SCL:
   IF #T.Now_M > #T.SP_M THEN #T.Now_M := #T.SP_M; END_IF;
END_REGION

REGION Network 5: Поправка переполнения секунд
   RUNG wire#powerrail
      { S7_Templates := "SrcType := Int" } EQ_Contact(in1 := #T.Now_M, in2 := #T.SP_M)
      { S7_Templates := "SrcType := Int" } GT_Contact(in1 := #T.Now_S, in2 := #T.SP_S)
      { S7_GenerateENO := "TRUE" } Move(in := #T.SP_S, out1 => #T.Now_S)
   END_RUNG
   // the same network as SCL:
   IF (#T.Now_M = #T.SP_M) AND (#T.Now_S > #T.SP_S) THEN #T.Now_S := #T.SP_S; END_IF;
END_REGION
END_FUNCTION

FUNCTION "Time_r" : Void   // FC106, LAD
{ S7_Optimized_Access := 'FALSE' }
VERSION : 0.1
   VAR_INPUT
      pulse : Bool;
   END_VAR
   VAR_IN_OUT
      C : Struct
         SP : Real;   // Уставка
         Now : Real;   // Текущий счёт
         One : Real;   // Вес импульса
         Progress : Real;   // Прогресс выполнения
         "Exit" : Bool;   // Счёт завершён
         Start : Bool;   // Запуск
         Pause : Bool;   // Пауза
         Reset : Bool;   // Сброс счёта
         pos : Bool;   // Контроль фронта сигнала
      END_STRUCT;
   END_VAR
   VAR_TEMP   // added for the SCL form of the ladder/FBD networks
      _w1 : Bool;
      _w2 : Bool;
   END_VAR
BEGIN

REGION Network 1: Подсчёт времени
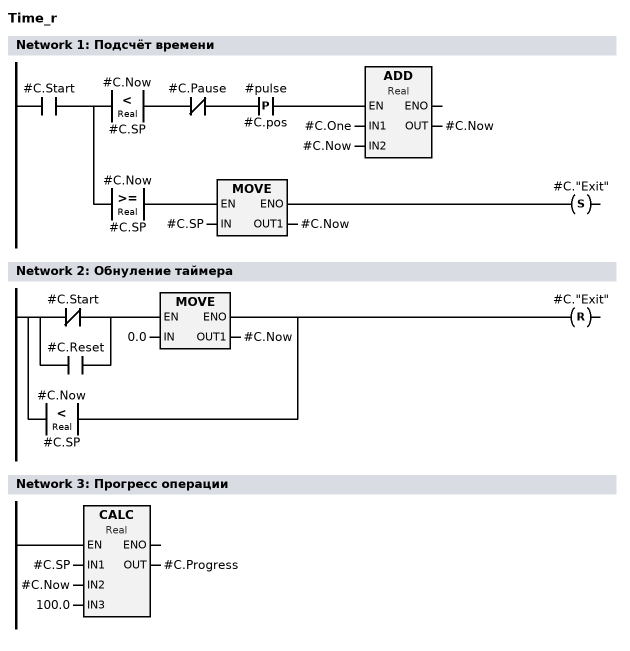
   RUNG wire#powerrail
      Contact( #C.Start )
      wire#w1
      { S7_Templates := "SrcType := Real" } LT_Contact(in1 := #C.Now, in2 := #C.SP)
      I_Contact( #C.Pause )
      P_Contact(operand := #pulse, bit := #C.pos)
      { S7_Templates := "SrcType := Real"; S7_GenerateENO := "TRUE" } Add(in1 := #C.One, in2 := #C.Now, out => #C.Now)
   END_RUNG
   RUNG wire#w1
      { S7_Templates := "SrcType := Real" } GE_Contact(in1 := #C.Now, in2 := #C.SP)
      Move(in := #C.SP, out1 => #C.Now)
      S_Coil( #C."Exit" )
   END_RUNG
   // the same network as SCL:
   #_w1 := #C.Start AND (#C.Now < #C.SP) AND NOT #C.Pause AND #pulse AND NOT #C.pos;   // rising edge of #pulse
   #C.pos := #pulse;
   IF #_w1 THEN #C.Now := #C.One + #C.Now; END_IF;
   #_w2 := #C.Start AND (#C.Now >= #C.SP);
   IF #_w2 THEN
       #C.Now := #C.SP;
       #C."Exit" := TRUE;
   END_IF;
END_REGION

REGION Network 2: Обнуление таймера
   RUNG wire#powerrail
      I_Contact( #C.Start )
      wire#w1
      { S7_GenerateENO := "TRUE" } Move(in := 0.0, out1 => #C.Now)
      wire#w2
      R_Coil( #C."Exit" )
   END_RUNG
   RUNG wire#powerrail
      Contact( #C.Reset )
   END_RUNG wire#w1
   RUNG wire#powerrail
      { S7_Templates := "SrcType := Real" } LT_Contact(in1 := #C.Now, in2 := #C.SP)
   END_RUNG wire#w2
   // the same network as SCL:
   // ENO of a box is taken as its EN; it also drops when the box reports an error
   #_w1 := NOT #C.Start OR #C.Reset;
   IF #_w1 THEN #C.Now := 0.0; END_IF;
   IF #_w1 OR (#C.Now < #C.SP) THEN #C."Exit" := FALSE; END_IF;
END_REGION

REGION Network 3: Прогресс операции
   CALC(in1 := #C.SP, in2 := #C.Now, in3 := 100.0, out => #C.Progress);
END_REGION
END_FUNCTION

FUNCTION "Time_as" : Void   // FC107, LAD
{ S7_Optimized_Access := 'FALSE' }
VERSION : 0.1
   VAR_INPUT
      Start : Bool;
      pulse : Bool;
   END_VAR
   VAR_IN_OUT
      Target : Real;
      Now : Real;
      T : Struct
         SP : Real;
         Now : Real;
         Dev : Real;
         Converter : Struct
            Use_Min_In : Bool;   // Отсекать входные значения ниже минимума
            Use_Max_In : Bool;   // Отсекать входные значения выше максимума
            Use_Min_Out : Bool;   // Отсекать результат ниже минимума
            Use_Max_Out : Bool;   // Отсекать результат выше максимума
            IO : Bool;   // Входной/Выходной режим
            Inverse : Bool;   // Инверсия выхода
            Min_In : Real;   // Минимальный входной сигнал
            Max_In : Real;   // Максимальный входной сигнал
            Min_Out : Real;   // Минимальный выходной сигнал
            Max_Out : Real;   // Максимальный выходной сигнал
         END_STRUCT;
         "Exit" : Bool;
         Start : Bool;
         Pause : Bool;
         sub : Bool;
         ok : Bool;
      END_STRUCT;
   END_VAR
   VAR_TEMP
      Max : Real;
      Min : Real;
   END_VAR
   VAR_TEMP   // added for the SCL form of the ladder/FBD networks
      _w1 : Bool;
      _w2 : Bool;
   END_VAR
BEGIN

REGION Network 1
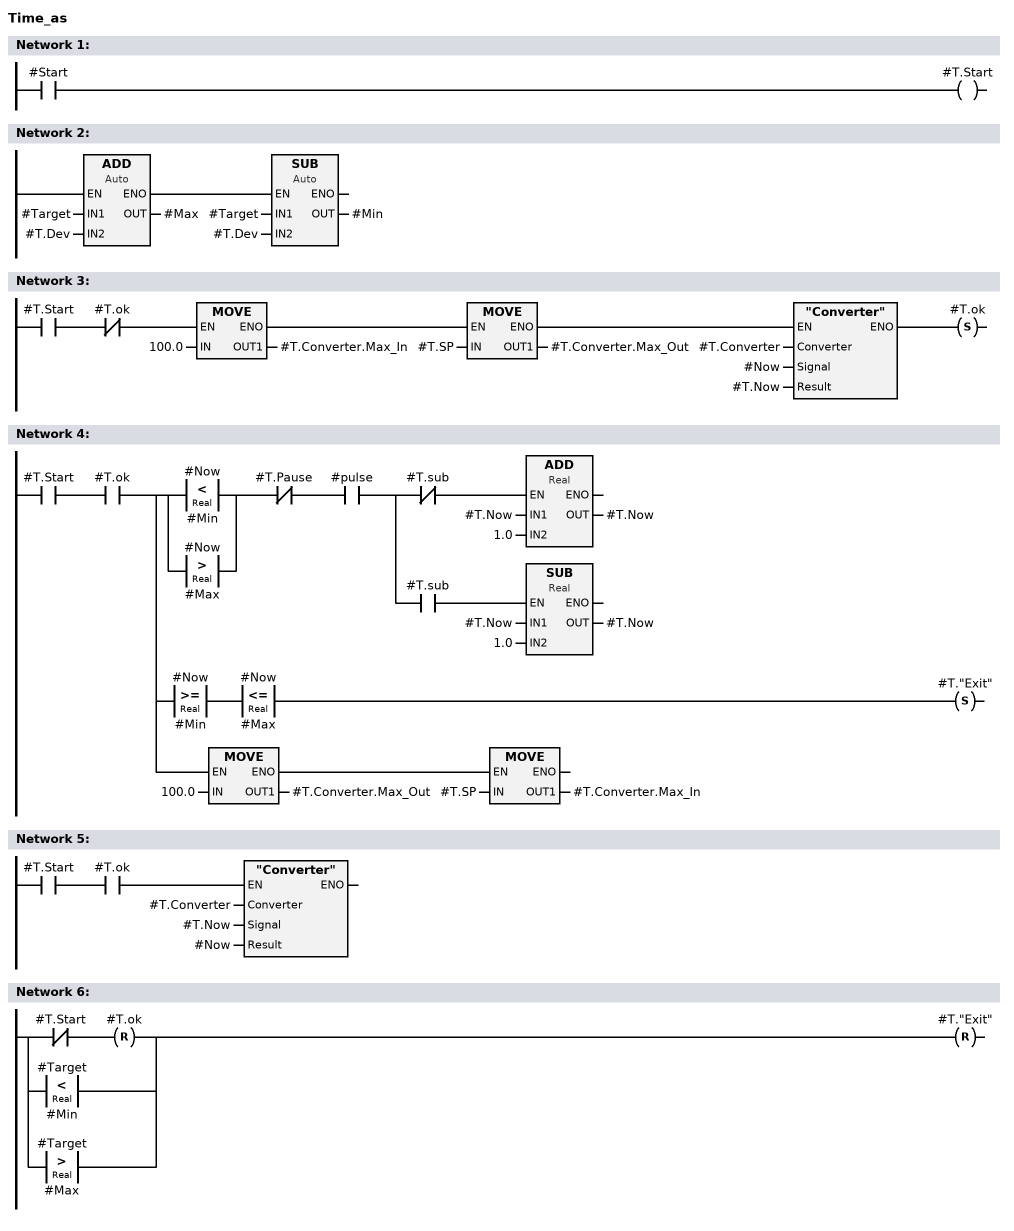
   RUNG wire#powerrail
      Contact( #Start )
      Coil( #T.Start )
   END_RUNG
   // the same network as SCL:
   #T.Start := #Start;
END_REGION

REGION Network 2
   RUNG wire#powerrail
      Add(in1 := #Target, in2 := #T.Dev, out => #Max)
      Sub(in1 := #Target, in2 := #T.Dev, out => #Min)
   END_RUNG
   // the same network as SCL:
   #Max := #Target + #T.Dev;
   #Min := #Target - #T.Dev;
END_REGION

REGION Network 3
   RUNG wire#powerrail
      Contact( #T.Start )
      I_Contact( #T.ok )
      Move(in := 100.0, out1 => #T.Converter.Max_In)
      Move(in := #T.SP, out1 => #T.Converter.Max_Out)
      "Converter"(Converter := #T.Converter, Signal := #Now, Result := #T.Now)
      S_Coil( #T.ok )
   END_RUNG
   // the same network as SCL:
   IF #T.Start AND NOT #T.ok THEN
       #T.Converter.Max_In := 100.0;
       #T.Converter.Max_Out := #T.SP;
   END_IF;
   "Converter"(EN := #T.Start AND NOT #T.ok,
               Converter := #T.Converter,
               Signal := #Now,
               Result := #T.Now,
               ENO => #_w1);
   IF #_w1 THEN #T.ok := TRUE; END_IF;
END_REGION

REGION Network 4
   RUNG wire#powerrail
      Contact( #T.Start )
      Contact( #T.ok )
      wire#w1
      { S7_Templates := "SrcType := Real" } LT_Contact(in1 := #Now, in2 := #Min)
      wire#w2
      I_Contact( #T.Pause )
      Contact( #pulse )
      wire#w3
      I_Contact( #T.sub )
      { S7_Templates := "SrcType := Real"; S7_GenerateENO := "TRUE" } Add(in1 := #T.Now, in2 := 1.0, out => #T.Now)
   END_RUNG
   RUNG wire#w1
      { S7_Templates := "SrcType := Real" } GT_Contact(in1 := #Now, in2 := #Max)
   END_RUNG wire#w2
   RUNG wire#w3
      Contact( #T.sub )
      { S7_Templates := "SrcType := Real"; S7_GenerateENO := "TRUE" } Sub(in1 := #T.Now, in2 := 1.0, out => #T.Now)
   END_RUNG
   RUNG wire#w1
      { S7_Templates := "SrcType := Real" } GE_Contact(in1 := #Now, in2 := #Min)
      { S7_Templates := "SrcType := Real" } LE_Contact(in1 := #Now, in2 := #Max)
      S_Coil( #T."Exit" )
   END_RUNG
   RUNG wire#w1
      Move(in := 100.0, out1 => #T.Converter.Max_Out)
      Move(in := #T.SP, out1 => #T.Converter.Max_In)
   END_RUNG
   // the same network as SCL:
   #_w1 := #T.Start AND #T.ok;
   #_w2 := #_w1 AND ((#Now < #Min) OR (#Now > #Max)) AND NOT #T.Pause AND #pulse;
   IF #_w2 AND NOT #T.sub THEN #T.Now := #T.Now + 1.0; END_IF;
   IF #_w2 AND #T.sub THEN #T.Now := #T.Now - 1.0; END_IF;
   IF #_w1 AND (#Now >= #Min) AND (#Now <= #Max) THEN #T."Exit" := TRUE; END_IF;
   IF #_w1 THEN
       #T.Converter.Max_Out := 100.0;
       #T.Converter.Max_In := #T.SP;
   END_IF;
END_REGION

REGION Network 5
   RUNG wire#powerrail
      Contact( #T.Start )
      Contact( #T.ok )
      "Converter"(Converter := #T.Converter, Signal := #T.Now, Result := #Now)
   END_RUNG
   // the same network as SCL:
   IF #T.Start AND #T.ok THEN
       "Converter"(Converter := #T.Converter, Signal := #T.Now, Result := #Now);
   END_IF;
END_REGION

REGION Network 6
   RUNG wire#powerrail
      I_Contact( #T.Start )
      R_Coil( #T.ok )
      wire#w1
      R_Coil( #T."Exit" )
   END_RUNG
   RUNG wire#powerrail
      { S7_Templates := "SrcType := Real" } LT_Contact(in1 := #Target, in2 := #Min)
   END_RUNG wire#w1
   RUNG wire#powerrail
      { S7_Templates := "SrcType := Real" } GT_Contact(in1 := #Target, in2 := #Max)
   END_RUNG wire#w1
   // the same network as SCL:
   IF NOT #T.Start THEN #T.ok := FALSE; END_IF;
   IF NOT #T.Start OR (#Target < #Min) OR (#Target > #Max) THEN #T."Exit" := FALSE; END_IF;
END_REGION
END_FUNCTION

FUNCTION "PLF_FC" : Void   // FC109, SCL
{ S7_Optimized_Access := 'TRUE' }
VERSION : 0.1
   VAR_INPUT
      REQ : Real;   // Запрошенная производительность
   END_VAR
   VAR_IN_OUT
      Now : Bool;   // Блок активен
      PLF_1 : Struct
         Use : Bool;
         Low : Real;   // Диапазон ОТ
         High : Real;   // Диапазон ДО
         Point_A : Real;   // Команда ОТ
         Point_B : Real;   // Команда ДО
         res : Word;
      END_STRUCT;
      PLF_2 : Struct
         Use : Bool;
         Low : Real;   // Диапазон ОТ
         High : Real;   // Диапазон ДО
         Point_A : Real;   // Команда ОТ
         Point_B : Real;   // Команда ДО
         res : Word;
      END_STRUCT;
      SP : Real;
   END_VAR
BEGIN
   // передаём стартовые точки в следующий фрагмент
   #PLF_2.Low := #PLF_1.High;
   #PLF_2.Point_A := #PLF_1.Point_B;

   // отключаем при некорректных значениях
   IF #PLF_1.High <= #PLF_1.Low OR #PLF_1.Point_B < #PLF_1.Point_B THEN
       #PLF_1.Use := False;
   END_IF;

   // отключаем при неполном графике
   IF #PLF_2.Use AND NOT #PLF_1.Use THEN
       #PLF_2.Use := False;
   END_IF;

   // следующий фрагмент используется 
   IF #PLF_1.Use AND #PLF_2.Use AND #REQ > #PLF_1.Low AND #REQ <= #PLF_1.High THEN
       #SP := ((#REQ - #PLF_1.Low) / ((#PLF_1.High - #PLF_1.Low) / (#PLF_1.Point_B - #PLF_1.Point_A))) + #PLF_1.Point_A;
       #Now := True;
   END_IF;

   // следующий фрагмент не задействован
   IF #PLF_1.Use AND NOT #PLF_2.Use AND #REQ > #PLF_1.Low THEN
       IF #REQ <= #PLF_1.High THEN
           #SP := ((#REQ - #PLF_1.Low) / ((#PLF_1.High - #PLF_1.Low) / (#PLF_1.Point_B - #PLF_1.Point_A))) + #PLF_1.Point_A;
       END_IF;
       IF #REQ > #PLF_1.High THEN
           #SP := #PLF_1.Point_B;
       END_IF;
       #Now := True;
   END_IF;

   // фрагмент не активен
   IF NOT #PLF_1.Use OR #REQ <= #PLF_1.Low OR (#PLF_1.Use AND #PLF_2.Use AND #REQ > #PLF_1.High) THEN
       #Now := False;
   END_IF;
END_FUNCTION

FUNCTION "R_to_T" : Void   // FC110, LAD
{ S7_Optimized_Access := 'TRUE' }
VERSION : 0.1
   VAR_INPUT
      R : Real;   // Время в секундах
   END_VAR
   VAR_OUTPUT
      T : Time;   // Время
   END_VAR
   VAR_TEMP
      D : DInt;   // Буфер
   END_VAR
BEGIN

REGION Network 1: Конвертация REAL to Time
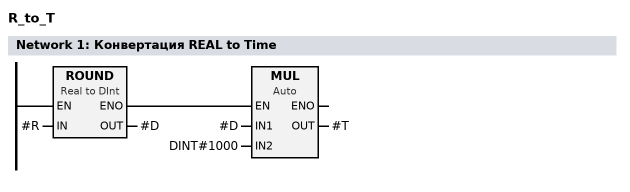
   RUNG wire#powerrail
      { S7_Templates := "[SrcType := Real, DestType := DInt]" } Round(in := #R, out => #D)
      Mul(in1 := #D, in2 := DINT#1000, out => #T)
   END_RUNG
   // the same network as SCL:
   #D := ROUND(#R);
   #T := #D * DINT#1000;
END_REGION
END_FUNCTION

FUNCTION "INV" : Void   // FC111, LAD
{ S7_Optimized_Access := 'TRUE' }
VERSION : 0.1
   VAR_INPUT
      S : Bool;   // Сигнал
      I : Bool;   // Инверсия
   END_VAR
   VAR_IN_OUT
      R : Bool;   // Результат
   END_VAR
BEGIN

REGION Network 1: Инверсия сигнала
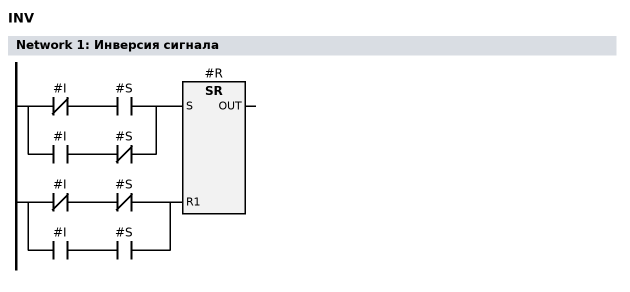
   RUNG wire#powerrail
      I_Contact( #I )
      Contact( #S )
      wire#w1
      S_SR(operand := #R, r1 := wire#w2)
   END_RUNG
   RUNG wire#powerrail
      Contact( #I )
      I_Contact( #S )
   END_RUNG wire#w1
   RUNG wire#powerrail
      I_Contact( #I )
      I_Contact( #S )
   END_RUNG wire#w2
   RUNG wire#powerrail
      Contact( #I )
      Contact( #S )
   END_RUNG wire#w2
   // the same network as SCL:
   IF (NOT #I AND #S) OR (#I AND NOT #S) THEN
       #R := TRUE;   // SR flip-flop
   END_IF;
   IF (NOT #I AND NOT #S) OR (#I AND #S) THEN #R := FALSE; END_IF;
END_REGION
END_FUNCTION

FUNCTION "ASCII to Int" : Void   // FC112, LAD
{ S7_Optimized_Access := 'TRUE' }
VERSION : 0.1
   VAR_INPUT
      Code : Word;
   END_VAR
   VAR_OUTPUT
      Symbol : Int;
   END_VAR
BEGIN

REGION Network 1
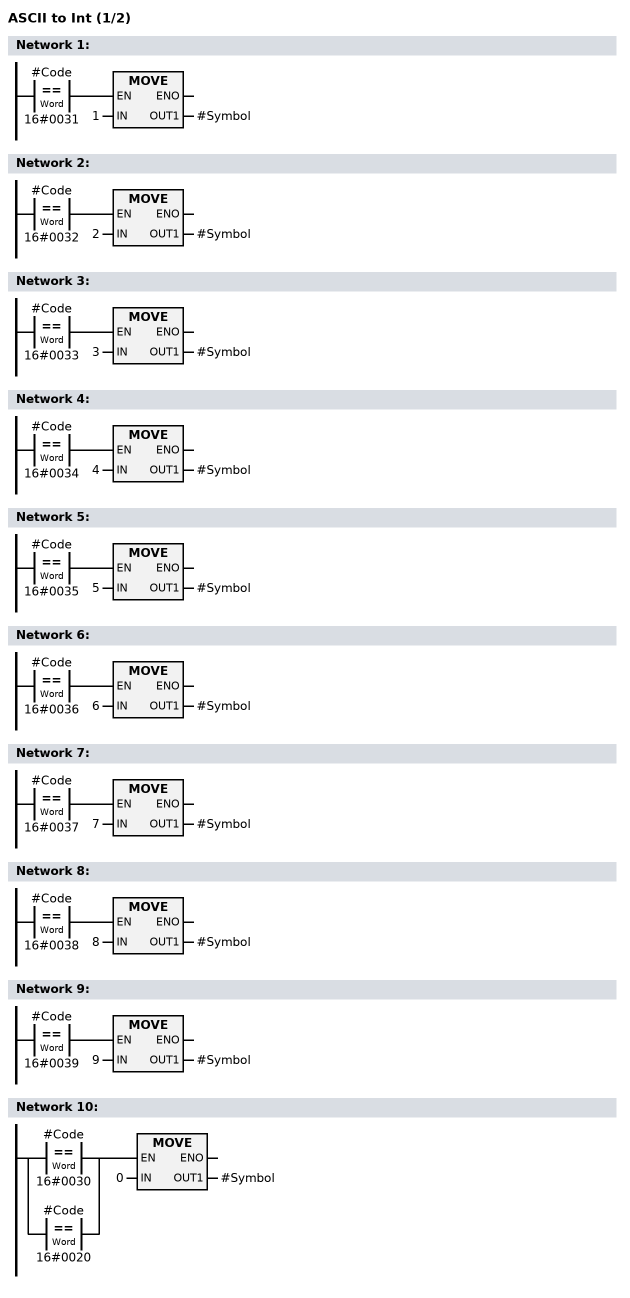
   RUNG wire#powerrail
      { S7_Templates := "SrcType := Word" } EQ_Contact(in1 := #Code, in2 := 16#0031)
      Move(in := 1, out1 => #Symbol)
   END_RUNG
   // the same network as SCL:
   IF #Code = 16#0031 THEN #Symbol := 1; END_IF;
END_REGION

REGION Network 2
   RUNG wire#powerrail
      { S7_Templates := "SrcType := Word" } EQ_Contact(in1 := #Code, in2 := 16#0032)
      Move(in := 2, out1 => #Symbol)
   END_RUNG
   // the same network as SCL:
   IF #Code = 16#0032 THEN #Symbol := 2; END_IF;
END_REGION

REGION Network 3
   RUNG wire#powerrail
      { S7_Templates := "SrcType := Word" } EQ_Contact(in1 := #Code, in2 := 16#0033)
      Move(in := 3, out1 => #Symbol)
   END_RUNG
   // the same network as SCL:
   IF #Code = 16#0033 THEN #Symbol := 3; END_IF;
END_REGION

REGION Network 4
   RUNG wire#powerrail
      { S7_Templates := "SrcType := Word" } EQ_Contact(in1 := #Code, in2 := 16#0034)
      Move(in := 4, out1 => #Symbol)
   END_RUNG
   // the same network as SCL:
   IF #Code = 16#0034 THEN #Symbol := 4; END_IF;
END_REGION

REGION Network 5
   RUNG wire#powerrail
      { S7_Templates := "SrcType := Word" } EQ_Contact(in1 := #Code, in2 := 16#0035)
      Move(in := 5, out1 => #Symbol)
   END_RUNG
   // the same network as SCL:
   IF #Code = 16#0035 THEN #Symbol := 5; END_IF;
END_REGION

REGION Network 6
   RUNG wire#powerrail
      { S7_Templates := "SrcType := Word" } EQ_Contact(in1 := #Code, in2 := 16#0036)
      Move(in := 6, out1 => #Symbol)
   END_RUNG
   // the same network as SCL:
   IF #Code = 16#0036 THEN #Symbol := 6; END_IF;
END_REGION

REGION Network 7
   RUNG wire#powerrail
      { S7_Templates := "SrcType := Word" } EQ_Contact(in1 := #Code, in2 := 16#0037)
      Move(in := 7, out1 => #Symbol)
   END_RUNG
   // the same network as SCL:
   IF #Code = 16#0037 THEN #Symbol := 7; END_IF;
END_REGION

REGION Network 8
   RUNG wire#powerrail
      { S7_Templates := "SrcType := Word" } EQ_Contact(in1 := #Code, in2 := 16#0038)
      Move(in := 8, out1 => #Symbol)
   END_RUNG
   // the same network as SCL:
   IF #Code = 16#0038 THEN #Symbol := 8; END_IF;
END_REGION

REGION Network 9
   RUNG wire#powerrail
      { S7_Templates := "SrcType := Word" } EQ_Contact(in1 := #Code, in2 := 16#0039)
      Move(in := 9, out1 => #Symbol)
   END_RUNG
   // the same network as SCL:
   IF #Code = 16#0039 THEN #Symbol := 9; END_IF;
END_REGION

REGION Network 10
   RUNG wire#powerrail
      { S7_Templates := "SrcType := Word" } EQ_Contact(in1 := #Code, in2 := 16#0030)
      wire#w1
      Move(in := 0, out1 => #Symbol)
   END_RUNG
   RUNG wire#powerrail
      { S7_Templates := "SrcType := Word" } EQ_Contact(in1 := #Code, in2 := 16#0020)
   END_RUNG wire#w1
   // the same network as SCL:
   IF (#Code = 16#0030) OR (#Code = 16#0020) THEN #Symbol := 0; END_IF;
END_REGION

REGION Network 11
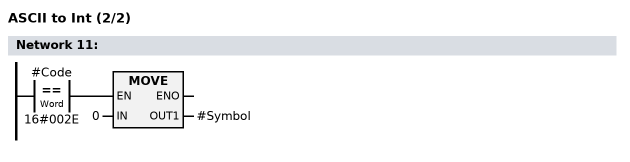
   RUNG wire#powerrail
      { S7_Templates := "SrcType := Word" } EQ_Contact(in1 := #Code, in2 := 16#002E)
      Move(in := 0, out1 => #Symbol)
   END_RUNG
   // the same network as SCL:
   IF #Code = 16#002E THEN #Symbol := 0; END_IF;
END_REGION
END_FUNCTION

FUNCTION "Mode" : Void   // FC150, LAD
{ S7_Optimized_Access := 'FALSE' }
VERSION : 0.1
   VAR_INPUT
      CMD : Struct   // Основные команды
         Hand : Bool;   // 0 - авто, 1 - ручной / 0 - Авто, 1 - Ручной
         Start_A : Bool;   // Автозапуск / Запуск в авторежиме
         Start_M : Bool;   // Ручной - вперёд / Запуск в ручном режиме
         Force : Bool;   // Принудительный
         Lock : Bool;   // Блокировать / Блокировка
         Local : Bool;   // Локальный
         Service : Bool;   // Сервис
         Safety : Bool;   // Безопасность
         Alarm : Bool;   // Есть авария / Авария
         Reset : Bool;   // Сброс аварий
         Sim : Bool;   // Режим симуляции
      END_STRUCT;
      All_Block : Bool;   // Аварийная блокировка
   END_VAR
   VAR_OUTPUT
      Mode : Int;   // Режим работы
   END_VAR
BEGIN

REGION Network 1: Автоматический режим
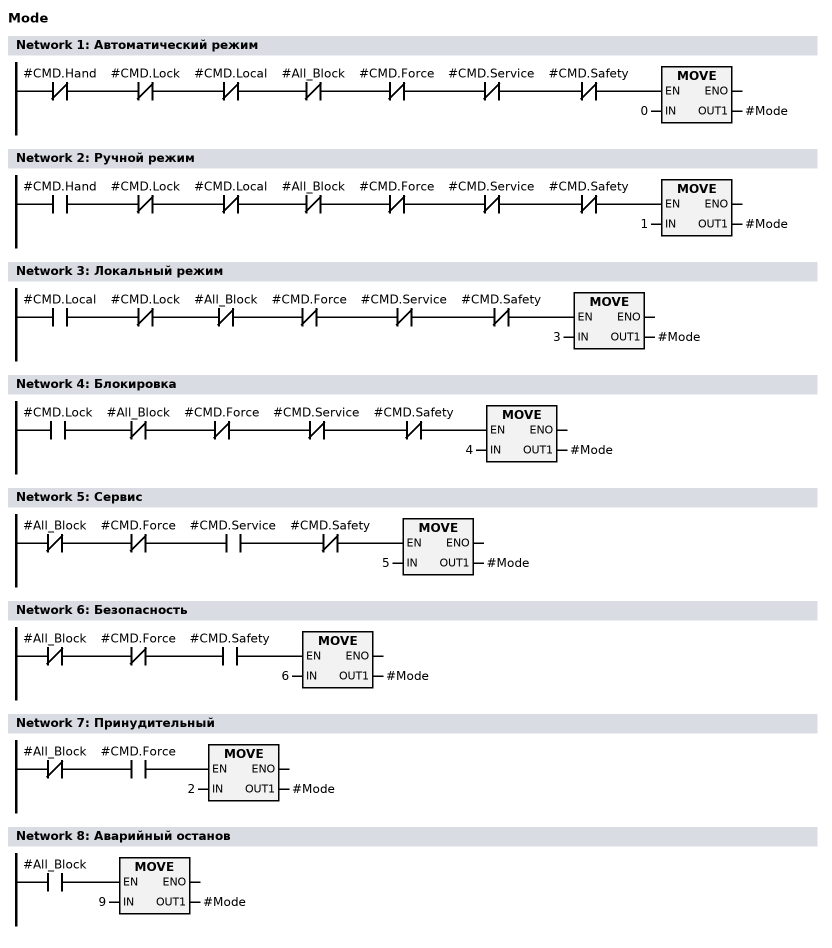
   RUNG wire#powerrail
      I_Contact( #CMD.Hand )
      I_Contact( #CMD.Lock )
      I_Contact( #CMD.Local )
      I_Contact( #All_Block )
      I_Contact( #CMD.Force )
      I_Contact( #CMD.Service )
      I_Contact( #CMD.Safety )
      { S7_GenerateENO := "TRUE" } Move(in := 0, out1 => #Mode)
   END_RUNG
   // the same network as SCL:
   IF NOT #CMD.Hand AND NOT #CMD.Lock AND NOT #CMD.Local AND NOT #All_Block AND NOT #CMD.Force AND NOT #CMD.Service AND NOT #CMD.Safety THEN
       #Mode := 0;
   END_IF;
END_REGION

REGION Network 2: Ручной режим
   RUNG wire#powerrail
      Contact( #CMD.Hand )
      I_Contact( #CMD.Lock )
      I_Contact( #CMD.Local )
      I_Contact( #All_Block )
      I_Contact( #CMD.Force )
      I_Contact( #CMD.Service )
      I_Contact( #CMD.Safety )
      { S7_GenerateENO := "TRUE" } Move(in := 1, out1 => #Mode)
   END_RUNG
   // the same network as SCL:
   IF #CMD.Hand AND NOT #CMD.Lock AND NOT #CMD.Local AND NOT #All_Block AND NOT #CMD.Force AND NOT #CMD.Service AND NOT #CMD.Safety THEN
       #Mode := 1;
   END_IF;
END_REGION

REGION Network 3: Локальный режим
   RUNG wire#powerrail
      Contact( #CMD.Local )
      I_Contact( #CMD.Lock )
      I_Contact( #All_Block )
      I_Contact( #CMD.Force )
      I_Contact( #CMD.Service )
      I_Contact( #CMD.Safety )
      { S7_GenerateENO := "TRUE" } Move(in := 3, out1 => #Mode)
   END_RUNG
   // the same network as SCL:
   IF #CMD.Local AND NOT #CMD.Lock AND NOT #All_Block AND NOT #CMD.Force AND NOT #CMD.Service AND NOT #CMD.Safety THEN
       #Mode := 3;
   END_IF;
END_REGION

REGION Network 4: Блокировка
   RUNG wire#powerrail
      Contact( #CMD.Lock )
      I_Contact( #All_Block )
      I_Contact( #CMD.Force )
      I_Contact( #CMD.Service )
      I_Contact( #CMD.Safety )
      { S7_GenerateENO := "TRUE" } Move(in := 4, out1 => #Mode)
   END_RUNG
   // the same network as SCL:
   IF #CMD.Lock AND NOT #All_Block AND NOT #CMD.Force AND NOT #CMD.Service AND NOT #CMD.Safety THEN
       #Mode := 4;
   END_IF;
END_REGION

REGION Network 5: Сервис
   RUNG wire#powerrail
      I_Contact( #All_Block )
      I_Contact( #CMD.Force )
      Contact( #CMD.Service )
      I_Contact( #CMD.Safety )
      { S7_GenerateENO := "TRUE" } Move(in := 5, out1 => #Mode)
   END_RUNG
   // the same network as SCL:
   IF NOT #All_Block AND NOT #CMD.Force AND #CMD.Service AND NOT #CMD.Safety THEN #Mode := 5; END_IF;
END_REGION

REGION Network 6: Безопасность
   RUNG wire#powerrail
      I_Contact( #All_Block )
      I_Contact( #CMD.Force )
      Contact( #CMD.Safety )
      { S7_GenerateENO := "TRUE" } Move(in := 6, out1 => #Mode)
   END_RUNG
   // the same network as SCL:
   IF NOT #All_Block AND NOT #CMD.Force AND #CMD.Safety THEN #Mode := 6; END_IF;
END_REGION

REGION Network 7: Принудительный
   RUNG wire#powerrail
      I_Contact( #All_Block )
      Contact( #CMD.Force )
      { S7_GenerateENO := "TRUE" } Move(in := 2, out1 => #Mode)
   END_RUNG
   // the same network as SCL:
   IF NOT #All_Block AND #CMD.Force THEN #Mode := 2; END_IF;
END_REGION

REGION Network 8: Аварийный останов
   RUNG wire#powerrail
      Contact( #All_Block )
      { S7_GenerateENO := "TRUE" } Move(in := 9, out1 => #Mode)
   END_RUNG
   // the same network as SCL:
   IF #All_Block THEN #Mode := 9; END_IF;
END_REGION
END_FUNCTION

// folder: statistic

FUNCTION_BLOCK "move_stat"   // FB13, LAD
{ S7_Optimized_Access := 'FALSE' }
VERSION : 0.1
   VAR
      In_the_beggin : Bool;
      down : Bool;
      up : Bool;
      box_weight : Array[1..25] of Real;
      box : Array[1..25] of Int;
      func_reset_Instance : "func_reset";
      func_down_Instance : "func_down";
      func_up_Instance : "func_up";
   END_VAR
   VAR_TEMP   // added for the SCL form of the ladder/FBD networks
      _w1 : Bool;
   END_VAR
   // box[1] := 1;
   // box[2] := 2;
   // box[3] := 3;
   // box[4] := 4;
   // box[5] := 5;
   // box[6] := 6;
   // box[7] := 7;
   // box[8] := 8;
   // box[9] := 9;
   // box[10] := 10;
   // box[11] := 11;
   // box[12] := 12;
   // box[13] := 13;
   // box[14] := 14;
   // box[15] := 15;
   // box[16] := 16;
   // box[17] := 17;
   // box[18] := 18;
   // box[19] := 19;
   // box[20] := 20;
   // box[21] := 21;
   // box[22] := 22;
   // box[23] := 23;
   // box[24] := 24;
   // box[25] := 25;
   // box_weight[1] := 0.0;
   // box_weight[2] := 0.0;
   // box_weight[3] := 0.0;
   // box_weight[4] := 0.0;
   // box_weight[5] := 0.0;
   // box_weight[6] := 0.0;
   // box_weight[7] := 0.0;
   // box_weight[8] := 0.0;
   // box_weight[9] := 0.0;
   // box_weight[10] := 0.0;
   // box_weight[11] := 0.0;
   // box_weight[12] := 0.0;
   // box_weight[13] := 0.0;
   // box_weight[14] := 0.0;
   // box_weight[15] := 0.0;
   // box_weight[16] := 0.0;
   // box_weight[17] := 0.0;
   // box_weight[18] := 0.0;
   // box_weight[19] := 0.0;
   // box_weight[20] := 0.0;
   // box_weight[21] := 0.0;
   // box_weight[22] := 0.0;
   // box_weight[23] := 0.0;
   // box_weight[24] := 0.0;
   // box_weight[25] := 0.0;
BEGIN

REGION Network 1
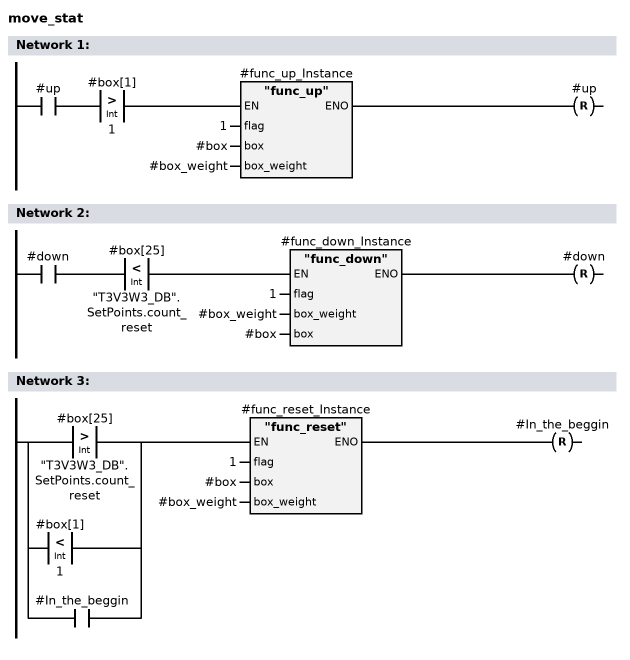
   RUNG wire#powerrail
      Contact( #up )
      { S7_Templates := "SrcType := Int" } GT_Contact(in1 := #box[1], in2 := 1)
      #func_up_Instance(flag := 1, box := #box, box_weight := #box_weight)
      R_Coil( #up )
   END_RUNG
   // the same network as SCL:
   #func_up_Instance(EN := #up AND (#box[1] > 1),   // "func_up"
                     flag := 1,
                     box := #box,
                     box_weight := #box_weight,
                     ENO => #_w1);
   IF #_w1 THEN #up := FALSE; END_IF;
END_REGION

REGION Network 2
   RUNG wire#powerrail
      Contact( #down )
      { S7_Templates := "SrcType := Int" } LT_Contact(in1 := #box[25], in2 := "T3V3W3_DB".SetPoints.count_reset)
      #func_down_Instance(flag := 1, box_weight := #box_weight, box := #box)
      R_Coil( #down )
   END_RUNG
   // the same network as SCL:
   #func_down_Instance(EN := #down AND (#box[25] < "T3V3W3_DB".SetPoints.count_reset),   // "func_down"
                       flag := 1,
                       box_weight := #box_weight,
                       box := #box,
                       ENO => #_w1);
   IF #_w1 THEN #down := FALSE; END_IF;
END_REGION

REGION Network 3
   RUNG wire#powerrail
      { S7_Templates := "SrcType := Int" } GT_Contact(in1 := #box[25], in2 := "T3V3W3_DB".SetPoints.count_reset)
      wire#w1
      #func_reset_Instance(flag := 1, box := #box, box_weight := #box_weight)
      R_Coil( #In_the_beggin )
   END_RUNG
   RUNG wire#powerrail
      { S7_Templates := "SrcType := Int" } LT_Contact(in1 := #box[1], in2 := 1)
   END_RUNG wire#w1
   RUNG wire#powerrail
      Contact( #In_the_beggin )
   END_RUNG wire#w1
   // the same network as SCL:
   #func_reset_Instance(EN := (#box[25] > "T3V3W3_DB".SetPoints.count_reset) OR (#box[1] < 1) OR #In_the_beggin,   // "func_reset"
                        flag := 1,
                        box := #box,
                        box_weight := #box_weight,
                        ENO => #_w1);
   IF #_w1 THEN #In_the_beggin := FALSE; END_IF;
END_REGION
END_FUNCTION_BLOCK

FUNCTION_BLOCK "Statistic"   // FB14, LAD
{ S7_Optimized_Access := 'FALSE' }
VERSION : 0.1
   VAR
      move_stat_Instance : "move_stat";
   END_VAR
   // move_stat_Instance.box_weight[1] := 0.0;
   // move_stat_Instance.box_weight[2] := 0.0;
   // move_stat_Instance.box_weight[11] := 0.0;
   // move_stat_Instance.box_weight[25] := 0.0;
   // move_stat_Instance.box_weight[24] := 0.0;
   // move_stat_Instance.box_weight[23] := 0.0;
   // move_stat_Instance.box_weight[21] := 0.0;
   // move_stat_Instance.box_weight[20] := 0.0;
   // move_stat_Instance.box_weight[19] := 0.0;
   // move_stat_Instance.box_weight[18] := 0.0;
   // move_stat_Instance.box_weight[17] := 0.0;
   // move_stat_Instance.box_weight[15] := 0.0;
   // move_stat_Instance.box_weight[14] := 0.0;
   // move_stat_Instance.box_weight[12] := 0.0;
   // move_stat_Instance.box_weight[22] := 0.0;
   // move_stat_Instance.box_weight[16] := 0.0;
   // move_stat_Instance.box_weight[13] := 0.0;
   // move_stat_Instance.box_weight[10] := 0.0;
   // move_stat_Instance.box_weight[9] := 0.0;
   // move_stat_Instance.box_weight[8] := 0.0;
   // move_stat_Instance.box_weight[7] := 0.0;
   // move_stat_Instance.box_weight[6] := 0.0;
   // move_stat_Instance.box_weight[5] := 0.0;
   // move_stat_Instance.box_weight[4] := 0.0;
   // move_stat_Instance.box_weight[3] := 0.0;
BEGIN

REGION Network 1
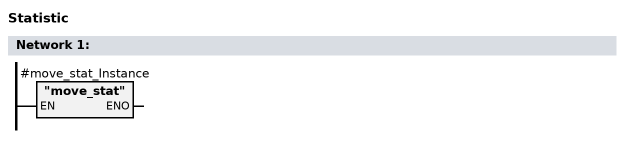
   RUNG wire#powerrail
      #move_stat_Instance()
   END_RUNG
   // the same network as SCL:
   #move_stat_Instance();   // "move_stat"
END_REGION
END_FUNCTION_BLOCK

FUNCTION_BLOCK "func_up"   // FB15, SCL
{ S7_Optimized_Access := 'FALSE' }
VERSION : 0.1
   VAR_INPUT
      flag : Bool;
   END_VAR
   VAR_IN_OUT
      box : Array[1..25] of Int;
      box_weight : Array[1..25] of Real;
   END_VAR
   VAR
      i : Int;
   END_VAR
BEGIN
   IF #flag = 1 THEN
       FOR #i := 1 TO 25 DO // Statement section IF
           #box[#i] := #box[#i] - 25;
           #box_weight[#i] := "bd".weight_box[#box[#i]];
       END_FOR;
   END_IF;
END_FUNCTION_BLOCK

FUNCTION_BLOCK "func_down"   // FB16, SCL
{ S7_Optimized_Access := 'FALSE' }
VERSION : 0.1
   VAR_INPUT
      flag : Bool;
   END_VAR
   VAR_IN_OUT
      box_weight : Array[1..25] of Real;
      box : Array[1..25] of Int;
   END_VAR
   VAR
      i : Int;
   END_VAR
BEGIN
   IF #flag = 1 THEN
       FOR #i := 1 TO 25 DO // Statement section IF
           #box[#i] := #box[#i] + 25;
           #box_weight[#i] := "bd".weight_box[#box[#i]];
       END_FOR;
       #flag := 0;
   END_IF;
END_FUNCTION_BLOCK

FUNCTION_BLOCK "func_reset"   // FB17, SCL
{ S7_Optimized_Access := 'FALSE' }
VERSION : 0.1
   VAR_INPUT
      flag : Bool;
   END_VAR
   VAR_IN_OUT
      box : Array[1..25] of Int;
      box_weight : Array[1..25] of Real;
   END_VAR
   VAR
      i : Int;
   END_VAR
BEGIN
   IF #flag = 1 THEN
       FOR #i := 1 TO 25 DO // Statement section IF
           #box[#i] := #i;
           #box_weight[#i] := "bd".weight_box[#box[#i]];
       END_FOR;
       #flag := 0;
   END_IF;
END_FUNCTION_BLOCK

FUNCTION_BLOCK "Reset_st"   // FB18, SCL
{ S7_Optimized_Access := 'FALSE' }
VERSION : 0.1
   VAR_INPUT
      flag : Bool;
   END_VAR
   VAR
      k : Real;
      i : Int;
   END_VAR
BEGIN
       IF #flag = 1 THEN
           FOR #i := 1 TO "T3V3W3_DB".SetPoints.count_reset DO // Statement section IF
             "bd".weight_box[#i] := #k;
           END_FOR;
           #flag := 0;
       END_IF;
END_FUNCTION_BLOCK

(* ===== HMI "HMI_RT_2" =====
system functions are stored by id; their names below are inferred from use
connection "HMI_Connection_2": ETHERNET, S7_1200_OMS

HMI tags "Standard-Variablentabelle"
   "WP231PR_DB_DR03_RESERVED_130" : String[12] = PLC WP231PR_DB.DR03.RESERVED_130 AT %DB231.DBX662.0, 1 s

HMI tags "Data Record DR3"
   "WP231PR_DB_DR03_SCALE_NAME" : String[12] = PLC WP231PR_DB.DR03.SCALE_NAME AT %DB231.DBX542.0, 1 s
   "WP231PR_DB_DR03_WEIGHT_UNIT" : String[4] = PLC WP231PR_DB.DR03.WEIGHT_UNIT AT %DB231.DBX556.0, 1 s
   "WP231PR_DB_DR03_LETTER_GROSS_WEIGHT_2" : Byte = PLC WP231PR_DB.DR03.LETTER_GROSS_WEIGHT_2 AT %DB231.DBB565, 1 s
   "WP231PR_DB_DR03_RESTRICTION_CODE" : UInt = PLC WP231PR_DB.DR03.RESTRICTION_CODE AT %DB231.DBW568, 1 s
   "WP231PR_DB_DR03_MIN_WEIGHT_D" : UInt = PLC WP231PR_DB.DR03.MIN_WEIGHT_D AT %DB231.DBW570, 1 s
   "WP231PR_DB_DR03_MAX_WEIGHT" : Real = PLC WP231PR_DB.DR03.MAX_WEIGHT AT %DB231.DBD574, 1 s
   "WP231PR_DB_DR03_CALIB_WEIGHT_0" : Real = PLC WP231PR_DB.DR03.CALIB_WEIGHT_0 AT %DB231.DBD578, 1 s
   "WP231PR_DB_DR03_CALIB_WEIGHT_1" : Real = PLC WP231PR_DB.DR03.CALIB_WEIGHT_1 AT %DB231.DBD582, 1 s
   "WP231PR_DB_DR03_CALIB_WEIGHT_2" : Real = PLC WP231PR_DB.DR03.CALIB_WEIGHT_2 AT %DB231.DBD586, 1 s
   "WP231PR_DB_DR03_CALIB_DIGITS_0" : DInt = PLC WP231PR_DB.DR03.CALIB_DIGITS_0 AT %DB231.DBD590, 1 s
   "WP231PR_DB_DR03_CALIB_DIGITS_1" : DInt = PLC WP231PR_DB.DR03.CALIB_DIGITS_1 AT %DB231.DBD594, 1 s
   "WP231PR_DB_DR03_CALIB_DIGITS_2" : DInt = PLC WP231PR_DB.DR03.CALIB_DIGITS_2 AT %DB231.DBD598, 1 s
   "WP231PR_DB_DR03_RESOLUTION_D" : Real = PLC WP231PR_DB.DR03.RESOLUTION_D AT %DB231.DBD602, 1 s
   "WP231PR_DB_DR03_INITIAL_ZEROING" : Bool = PLC WP231PR_DB.DR03.INITIAL_ZEROING AT %DB231.DBX607.0, 1 s
   "WP231PR_DB_DR03_INITIAL_ZEROING_IF_TARED" : Bool = PLC WP231PR_DB.DR03.INITIAL_ZEROING_IF_TARED AT %DB231.DBX607.1, 1 s
   "WP231PR_DB_DR03_ZERO_TRACKING" : Bool = PLC WP231PR_DB.DR03.ZERO_TRACKING AT %DB231.DBX607.2, 1 s
   "WP231PR_DB_DR03_ADDITIVE_TARE" : Bool = PLC WP231PR_DB.DR03.ADDITIVE_TARE AT %DB231.DBX607.3, 1 s
   "WP231PR_DB_DR03_WEIGHT_SIM_ALLOWED" : Bool = PLC WP231PR_DB.DR03.WEIGHT_SIM_ALLOWED AT %DB231.DBX607.4, 1 s
   "WP231PR_DB_DR03_DEC_POINT_PROC_VAL" : UInt = PLC WP231PR_DB.DR03.DEC_POINT_PROC_VAL AT %DB231.DBW608, 1 s
   "WP231PR_DB_DR03_TARE_MAX" : Real = PLC WP231PR_DB.DR03.TARE_MAX AT %DB231.DBD610, 1 s
   "WP231PR_DB_DR03_INITIAL_ZEROING_LIM_NEG" : Real = PLC WP231PR_DB.DR03.INITIAL_ZEROING_LIM_NEG AT %DB231.DBD614, 1 s
   "WP231PR_DB_DR03_INITIAL_ZEROING_LIM_POS" : Real = PLC WP231PR_DB.DR03.INITIAL_ZEROING_LIM_POS AT %DB231.DBD618, 1 s
   "WP231PR_DB_DR03_SEM_AUT_ZERO_LIM_NEG" : Real = PLC WP231PR_DB.DR03.SEM_AUT_ZERO_LIM_NEG AT %DB231.DBD622, 1 s
   "WP231PR_DB_DR03_SEM_AUT_ZERO_LIM_POS" : Real = PLC WP231PR_DB.DR03.SEM_AUT_ZERO_LIM_POS AT %DB231.DBD626, 1 s
   "WP231PR_DB_DR03_ST_STILL_RANGE_D" : Real = PLC WP231PR_DB.DR03.ST_STILL_RANGE_D AT %DB231.DBD630, 1 s
   "WP231PR_DB_DR03_ST_STILL_TIME" : Time = PLC WP231PR_DB.DR03.ST_STILL_TIME AT %DB231.DBD634, 1 s
   "WP231PR_DB_DR03_ST_STILL_WAITING_TIME" : Time = PLC WP231PR_DB.DR03.ST_STILL_WAITING_TIME AT %DB231.DBD638, 1 s
   "WP231PR_DB_DR03_FREQ_LOW_PASS_1" : Real = PLC WP231PR_DB.DR03.FREQ_LOW_PASS_1 AT %DB231.DBD642, 1 s
   "WP231PR_DB_DR03_ORDER_NO_LOW_PASS_1" : UInt = PLC WP231PR_DB.DR03.ORDER_NO_LOW_PASS_1 AT %DB231.DBW646, 1 s
   "WP231PR_DB_DR03_FREQ_LOW_PASS_2" : Real = PLC WP231PR_DB.DR03.FREQ_LOW_PASS_2 AT %DB231.DBD650, 1 s
   "WP231PR_DB_DR03_ORDER_NO_LOW_PASS_2" : UInt = PLC WP231PR_DB.DR03.ORDER_NO_LOW_PASS_2 AT %DB231.DBW654, 1 s
   "WP231PR_DB_DR03_AVER_FILTER_DEPTH" : UInt = PLC WP231PR_DB.DR03.AVER_FILTER_DEPTH AT %DB231.DBW656, 1 s
   "WP231PR_DB_DR03_SHOW_WR_DATA" : UInt = PLC WP231PR_DB.DR03.SHOW_WR_DATA AT %DB231.DBW658, 1 s
   "WP231PR_DB_DR03_SECURE_DISPLAY_INTERFACE" : UInt = PLC WP231PR_DB.DR03.SECURE_DISPLAY_INTERFACE AT %DB231.DBW660, 1 s
   "WP231PR_DB_DR03_FW_VERSION_HMI_MODUL" : String[20] = PLC WP231PR_DB.DR03.FW_VERSION_HMI_MODUL AT %DB231.DBX698.0, 1 s
   "WP231PR_DB_DR03_MIN_ZOOMFACTOR" : UInt = PLC WP231PR_DB.DR03.MIN_ZOOMFACTOR AT %DB231.DBW720, 1 s

HMI tags "Data Record DR4"
   "WP231PR_DB_DR04_CALIB_DIGITS_0_CALC" : DInt = PLC WP231PR_DB.DR04.CALIB_DIGITS_0_CALC AT %DB231.DBD734, 1 s
   "WP231PR_DB_DR04_CALIB_DIGITS_1_CALC" : DInt = PLC WP231PR_DB.DR04.CALIB_DIGITS_1_CALC AT %DB231.DBD738, 1 s
   "WP231PR_DB_DR04_CALIB_DIGITS_2_CALC" : DInt = PLC WP231PR_DB.DR04.CALIB_DIGITS_2_CALC AT %DB231.DBD742, 1 s

HMI tags "Data Record DR5"
   "WP231PR_DB_DR05_TARE_WEIGHT_PRESET" : Real = PLC WP231PR_DB.DR05.TARE_WEIGHT_PRESET AT %DB231.DBD762, 1 s
   "WP231PR_DB_DR05_TARE_WEIGHT_SEM_AUT" : Real = PLC WP231PR_DB.DR05.TARE_WEIGHT_SEM_AUT AT %DB231.DBD766, 1 s
   "WP231PR_DB_DR05_ZEROING_WEIGHT_INITIAL" : Real = PLC WP231PR_DB.DR05.ZEROING_WEIGHT_INITIAL AT %DB231.DBD770, 1 s
   "WP231PR_DB_DR05_ZEROING_WEIGHT_SEM_AUT" : Real = PLC WP231PR_DB.DR05.ZEROING_WEIGHT_SEM_AUT AT %DB231.DBD774, 1 s
   "WP231PR_DB_DR05_ZEROING_WEIGHT_TRACKING" : Real = PLC WP231PR_DB.DR05.ZEROING_WEIGHT_TRACKING AT %DB231.DBD778, 1 s
   "WP231PR_DB_DR05_DEAD_LOAD" : Real = PLC WP231PR_DB.DR05.DEAD_LOAD AT %DB231.DBD782, 1 s

HMI tags "Data Record DR6"
   "WP231PR_DB_DR06_LIM_REFERENCE" : UInt = PLC WP231PR_DB.DR06.LIM_REFERENCE AT %DB231.DBW802, 1 s
   "WP231PR_DB_DR06_LIM_1_ON" : Real = PLC WP231PR_DB.DR06.LIM_1_ON AT %DB231.DBD806, 1 s
   "WP231PR_DB_DR06_DELAY_LIM_1_ON" : Time = PLC WP231PR_DB.DR06.DELAY_LIM_1_ON AT %DB231.DBD810, 1 s
   "WP231PR_DB_DR06_LIM_1_OFF" : Real = PLC WP231PR_DB.DR06.LIM_1_OFF AT %DB231.DBD814, 1 s
   "WP231PR_DB_DR06_DELAY_LIM_1_OFF" : Time = PLC WP231PR_DB.DR06.DELAY_LIM_1_OFF AT %DB231.DBD818, 1 s
   "WP231PR_DB_DR06_LIM_2_ON" : Real = PLC WP231PR_DB.DR06.LIM_2_ON AT %DB231.DBD822, 1 s
   "WP231PR_DB_DR06_DELAY_LIM_2_ON" : Time = PLC WP231PR_DB.DR06.DELAY_LIM_2_ON AT %DB231.DBD826, 1 s
   "WP231PR_DB_DR06_LIM_2_OFF" : Real = PLC WP231PR_DB.DR06.LIM_2_OFF AT %DB231.DBD830, 1 s
   "WP231PR_DB_DR06_DELAY_LIM_2_OFF" : Time = PLC WP231PR_DB.DR06.DELAY_LIM_2_OFF AT %DB231.DBD834, 1 s
   "WP231PR_DB_DR06_LIMIT_3_EMPTY" : Real = PLC WP231PR_DB.DR06.LIMIT_3_EMPTY AT %DB231.DBD838, 1 s
   "WP231PR_DB_DR06_DELAY_EMPTY" : Time = PLC WP231PR_DB.DR06.DELAY_EMPTY AT %DB231.DBD842, 1 s

HMI tags "Data Record DR7"
   "WP231PR_DB_DR07_ASSIGN_DI_0" : UInt = PLC WP231PR_DB.DR07.ASSIGN_DI_0 AT %DB231.DBW862, 1 s
   "WP231PR_DB_DR07_ASSIGN_DI_1" : UInt = PLC WP231PR_DB.DR07.ASSIGN_DI_1 AT %DB231.DBW864, 1 s
   "WP231PR_DB_DR07_ASSIGN_DI_2" : UInt = PLC WP231PR_DB.DR07.ASSIGN_DI_2 AT %DB231.DBW866, 1 s
   "WP231PR_DB_DR07_ASSIGN_DI_3" : UInt = PLC WP231PR_DB.DR07.ASSIGN_DI_3 AT %DB231.DBW868, 1 s
   "WP231PR_DB_DR07_FILTER_DI" : UInt = PLC WP231PR_DB.DR07.FILTER_DI AT %DB231.DBW870, 1 s
   "WP231PR_DB_DR07_ASSIGN_DQ_0" : UInt = PLC WP231PR_DB.DR07.ASSIGN_DQ_0 AT %DB231.DBW872, 1 s
   "WP231PR_DB_DR07_ASSIGN_DQ_1" : UInt = PLC WP231PR_DB.DR07.ASSIGN_DQ_1 AT %DB231.DBW874, 1 s
   "WP231PR_DB_DR07_ASSIGN_DQ_2" : UInt = PLC WP231PR_DB.DR07.ASSIGN_DQ_2 AT %DB231.DBW876, 1 s
   "WP231PR_DB_DR07_ASSIGN_DQ_3" : UInt = PLC WP231PR_DB.DR07.ASSIGN_DQ_3 AT %DB231.DBW878, 1 s
   "WP231PR_DB_DR07_ANA_OUT_BY_ERR_OR_STOP" : UInt = PLC WP231PR_DB.DR07.ANA_OUT_BY_ERR_OR_STOP AT %DB231.DBW880, 1 s
   "WP231PR_DB_DR07_DQ_0_BY_ERR_OR_STOP" : Bool = PLC WP231PR_DB.DR07.DQ_0_BY_ERR_OR_STOP AT %DB231.DBX883.0, 1 s
   "WP231PR_DB_DR07_DQ_1_BY_ERR_OR_STOP" : Bool = PLC WP231PR_DB.DR07.DQ_1_BY_ERR_OR_STOP AT %DB231.DBX883.1, 1 s
   "WP231PR_DB_DR07_DQ_2_BY_ERR_OR_STOP" : Bool = PLC WP231PR_DB.DR07.DQ_2_BY_ERR_OR_STOP AT %DB231.DBX883.2, 1 s
   "WP231PR_DB_DR07_DQ_3_BY_ERR_OR_STOP" : Bool = PLC WP231PR_DB.DR07.DQ_3_BY_ERR_OR_STOP AT %DB231.DBX883.3, 1 s
   "WP231PR_DB_DR07_RANGE_ANA_OUT" : UInt = PLC WP231PR_DB.DR07.RANGE_ANA_OUT AT %DB231.DBW884, 1 s
   "WP231PR_DB_DR07_SOURCE_ANA_OUT" : UInt = PLC WP231PR_DB.DR07.SOURCE_ANA_OUT AT %DB231.DBW886, 1 s
   "WP231PR_DB_DR07_ANA_OUT_BY_ERR_OR_STOP_1" : UInt = PLC WP231PR_DB.DR07.ANA_OUT_BY_ERR_OR_STOP_1 AT %DB231.DBW888, 1 s
   "WP231PR_DB_DR07_START_VAL_ANA_OUT" : Real = PLC WP231PR_DB.DR07.START_VAL_ANA_OUT AT %DB231.DBD890, 1 s
   "WP231PR_DB_DR07_END_VAL_ANA_OUT" : Real = PLC WP231PR_DB.DR07.END_VAL_ANA_OUT AT %DB231.DBD894, 1 s
   "WP231PR_DB_DR07_ANA_OUT_ERR" : Real = PLC WP231PR_DB.DR07.ANA_OUT_ERR AT %DB231.DBD898, 1 s
   "WP231PR_DB_DR07_TRACE_RATE" : UInt = PLC WP231PR_DB.DR07.TRACE_RATE AT %DB231.DBW902, 1 s
   "WP231PR_DB_DR07_TRACE_MEM_TYPE" : Bool = PLC WP231PR_DB.DR07.TRACE_MEM_TYPE AT %DB231.DBX905.0, 1 s

HMI tags "Data Record DR8"
   "WP231PR_DB_DR08_DATE_TIME" : DTL = PLC WP231PR_DB.DR08.DATE_TIME AT %DB231.DBX922.0, 1 s

HMI tags "Data Record DR9"
   "WP231PR_DB_DR09_ORDER_NO" : String[16] = PLC WP231PR_DB.DR09.ORDER_NO AT %DB231.DBX942.0, 1 s
   "WP231PR_DB_DR09_SERIAL_NO" : String[12] = PLC WP231PR_DB.DR09.SERIAL_NO AT %DB231.DBX960.0, 1 s
   "WP231PR_DB_DR09_FIRMWARE_VERS" : String[2] = PLC WP231PR_DB.DR09.FIRMWARE_VERS AT %DB231.DBX974.0, 1 s
   "WP231PR_DB_DR09_FIRMWARE_VERS_POS_1" : UInt = PLC WP231PR_DB.DR09.FIRMWARE_VERS_POS_1 AT %DB231.DBW978, 1 s
   "WP231PR_DB_DR09_FIRMWARE_VERS_POS_2" : UInt = PLC WP231PR_DB.DR09.FIRMWARE_VERS_POS_2 AT %DB231.DBW980, 1 s
   "WP231PR_DB_DR09_FIRMWARE_VERS_POS_3" : UInt = PLC WP231PR_DB.DR09.FIRMWARE_VERS_POS_3 AT %DB231.DBW982, 1 s
   "WP231PR_DB_DR09_HARDWARE_VERSION" : UInt = PLC WP231PR_DB.DR09.HARDWARE_VERSION AT %DB231.DBW984, 1 s
   "WP231PR_DB_DR09_OS_VERSION_2" : String[2] = PLC WP231PR_DB.DR09.OS_VERSION_2 AT %DB231.DBX986.0, 1 s
   "WP231PR_DB_DR09_OS_VERSION_1" : UInt = PLC WP231PR_DB.DR09.OS_VERSION_1 AT %DB231.DBW990, 1 s
   "WP231PR_DB_DR09_DRAM" : UInt = PLC WP231PR_DB.DR09.DRAM AT %DB231.DBW992, 1 s
   "WP231PR_DB_DR09_FLASH" : UInt = PLC WP231PR_DB.DR09.FLASH AT %DB231.DBW994, 1 s
   "WP231PR_DB_DR09_MRAM" : UInt = PLC WP231PR_DB.DR09.MRAM AT %DB231.DBW996, 1 s

HMI tags "Data Record DR10"
   "WP231PR_DB_DR10_NO_OF_LOAD_CELLS" : UInt = PLC WP231PR_DB.DR10.NO_OF_LOAD_CELLS AT %DB231.DBW1010, 1 s
   "WP231PR_DB_DR10_SWITCH_50_60_HZ" : UInt = PLC WP231PR_DB.DR10.SWITCH_50_60_HZ AT %DB231.DBW1012, 1 s
   "WP231PR_DB_DR10_NO_POINTS_OF_SUPPORT" : UInt = PLC WP231PR_DB.DR10.NO_POINTS_OF_SUPPORT AT %DB231.DBW1014, 1 s
   "WP231PR_DB_DR10_GAIN_LOAD_CELL" : Real = PLC WP231PR_DB.DR10.GAIN_LOAD_CELL AT %DB231.DBD1018, 1 s
   "WP231PR_DB_DR10_ZERO_OFFSET_LC" : Real = PLC WP231PR_DB.DR10.ZERO_OFFSET_LC AT %DB231.DBD1022, 1 s
   "WP231PR_DB_DR10_NOM_LOAD_ONE_LOAD_CELL" : Real = PLC WP231PR_DB.DR10.NOM_LOAD_ONE_LOAD_CELL AT %DB231.DBD1026, 1 s

HMI tags "Data Record DR12"
   "WP231PR_DB_DR12_DEVICE_MAC_ADDRESS" : UInt = PLC WP231PR_DB.DR12.DEVICE_MAC_ADDRESS AT %DB231.DBW1054, 1 s
   "WP231PR_DB_DR12_DEVICE_MAC_ADDRESS_1" : UInt = PLC WP231PR_DB.DR12.DEVICE_MAC_ADDRESS_1 AT %DB231.DBW1056, 1 s
   "WP231PR_DB_DR12_DEVICE_MAC_ADDRESS_2" : UInt = PLC WP231PR_DB.DR12.DEVICE_MAC_ADDRESS_2 AT %DB231.DBW1058, 1 s
   "WP231PR_DB_DR12_DEVICE_MAC_ADDRESS_3" : UInt = PLC WP231PR_DB.DR12.DEVICE_MAC_ADDRESS_3 AT %DB231.DBW1060, 1 s
   "WP231PR_DB_DR12_DEVICE_MAC_ADDRESS_4" : UInt = PLC WP231PR_DB.DR12.DEVICE_MAC_ADDRESS_4 AT %DB231.DBW1062, 1 s
   "WP231PR_DB_DR12_DEVICE_MAC_ADDRESS_5" : UInt = PLC WP231PR_DB.DR12.DEVICE_MAC_ADDRESS_5 AT %DB231.DBW1064, 1 s
   "WP231PR_DB_DR12_PORT_MAC_ADDRESS" : UInt = PLC WP231PR_DB.DR12.PORT_MAC_ADDRESS AT %DB231.DBW1066, 1 s
   "WP231PR_DB_DR12_PORT_MAC_ADDRESS_1" : UInt = PLC WP231PR_DB.DR12.PORT_MAC_ADDRESS_1 AT %DB231.DBW1068, 1 s
   "WP231PR_DB_DR12_PORT_MAC_ADDRESS_2" : UInt = PLC WP231PR_DB.DR12.PORT_MAC_ADDRESS_2 AT %DB231.DBW1070, 1 s
   "WP231PR_DB_DR12_PORT_MAC_ADDRESS_3" : UInt = PLC WP231PR_DB.DR12.PORT_MAC_ADDRESS_3 AT %DB231.DBW1072, 1 s
   "WP231PR_DB_DR12_PORT_MAC_ADDRESS_4" : UInt = PLC WP231PR_DB.DR12.PORT_MAC_ADDRESS_4 AT %DB231.DBW1074, 1 s
   "WP231PR_DB_DR12_PORT_MAC_ADDRESS_5" : UInt = PLC WP231PR_DB.DR12.PORT_MAC_ADDRESS_5 AT %DB231.DBW1076, 1 s
   "WP231PR_DB_DR12_IP_ADDRESS_1" : UInt = PLC WP231PR_DB.DR12.IP_ADDRESS_1 AT %DB231.DBW1078, 1 s
   "WP231PR_DB_DR12_IP_ADDRESS_2" : UInt = PLC WP231PR_DB.DR12.IP_ADDRESS_2 AT %DB231.DBW1080, 1 s
   "WP231PR_DB_DR12_IP_ADDRESS_3" : UInt = PLC WP231PR_DB.DR12.IP_ADDRESS_3 AT %DB231.DBW1082, 1 s
   "WP231PR_DB_DR12_IP_ADDRESS_4" : UInt = PLC WP231PR_DB.DR12.IP_ADDRESS_4 AT %DB231.DBW1084, 1 s
   "WP231PR_DB_DR12_SUB_NET_MASK_1" : UInt = PLC WP231PR_DB.DR12.SUB_NET_MASK_1 AT %DB231.DBW1086, 1 s
   "WP231PR_DB_DR12_SUB_NET_MASK_2" : UInt = PLC WP231PR_DB.DR12.SUB_NET_MASK_2 AT %DB231.DBW1088, 1 s
   "WP231PR_DB_DR12_SUB_NET_MASK_3" : UInt = PLC WP231PR_DB.DR12.SUB_NET_MASK_3 AT %DB231.DBW1090, 1 s
   "WP231PR_DB_DR12_SUB_NET_MASK_4" : UInt = PLC WP231PR_DB.DR12.SUB_NET_MASK_4 AT %DB231.DBW1092, 1 s
   "WP231PR_DB_DR12_CURRENT_GATEWAY_1" : UInt = PLC WP231PR_DB.DR12.CURRENT_GATEWAY_1 AT %DB231.DBW1094, 1 s
   "WP231PR_DB_DR12_CURRENT_GATEWAY_2" : UInt = PLC WP231PR_DB.DR12.CURRENT_GATEWAY_2 AT %DB231.DBW1096, 1 s
   "WP231PR_DB_DR12_CURRENT_GATEWAY_3" : UInt = PLC WP231PR_DB.DR12.CURRENT_GATEWAY_3 AT %DB231.DBW1098, 1 s
   "WP231PR_DB_DR12_CURRENT_GATEWAY_4" : UInt = PLC WP231PR_DB.DR12.CURRENT_GATEWAY_4 AT %DB231.DBW1100, 1 s

HMI tags "Data Record DR13"
   "WP231PR_DB_DR13_RS485_PROTOCOL" : UInt = PLC WP231PR_DB.DR13.RS485_PROTOCOL AT %DB231.DBW1154, 1 s
   "WP231PR_DB_DR13_RS485_BAUD_RATE" : UInt = PLC WP231PR_DB.DR13.RS485_BAUD_RATE AT %DB231.DBW1156, 1 s
   "WP231PR_DB_DR13_RS485_PARITY" : Bool = PLC WP231PR_DB.DR13.RS485_PARITY AT %DB231.DBX1159.0, 1 s
   "WP231PR_DB_DR13_RS485_DATA_BITS" : Bool = PLC WP231PR_DB.DR13.RS485_DATA_BITS AT %DB231.DBX1159.1, 1 s
   "WP231PR_DB_DR13_RS485_STOP_BITS" : Bool = PLC WP231PR_DB.DR13.RS485_STOP_BITS AT %DB231.DBX1159.2, 1 s
   "WP231PR_DB_DR13_MODBUS_RTU_ADDRESS" : UInt = PLC WP231PR_DB.DR13.MODBUS_RTU_ADDRESS AT %DB231.DBW1160, 1 s
   "WP231PR_DB_DR13_DEC_POINT_REM_DISPLAY" : Int = PLC WP231PR_DB.DR13.DEC_POINT_REM_DISPLAY AT %DB231.DBW1162, 1 s
   "WP231PR_DB_DR13_MODBUS_RTU_RESPONSE_DELAY" : UInt = PLC WP231PR_DB.DR13.MODBUS_RTU_RESPONSE_DELAY AT %DB231.DBW1164, 1 s

HMI tags "Data Record DR14"
   "WP231PR_DB_DR14_SEL_PROC_VAL_1_SIMATIC" : UInt = PLC WP231PR_DB.DR14.SEL_PROC_VAL_1_SIMATIC AT %DB231.DBW1178, 1 s
   "WP231PR_DB_DR14_SEL_PROC_VAL_2_SIMATIC" : UInt = PLC WP231PR_DB.DR14.SEL_PROC_VAL_2_SIMATIC AT %DB231.DBW1180, 1 s

HMI tags "Data Record DR15"
   "WP231PR_DB_DR15_PRESET_TARE_1" : Real = PLC WP231PR_DB.DR15.PRESET_TARE_1 AT %DB231.DBD1194, 1 s
   "WP231PR_DB_DR15_PRESET_TARE_2" : Real = PLC WP231PR_DB.DR15.PRESET_TARE_2 AT %DB231.DBD1198, 1 s
   "WP231PR_DB_DR15_PRESET_TARE_3" : Real = PLC WP231PR_DB.DR15.PRESET_TARE_3 AT %DB231.DBD1202, 1 s

HMI tags "Data Record DR16"
   "WP231PR_DB_DR16_SIMULATION_WEIGHT" : Real = PLC WP231PR_DB.DR16.SIMULATION_WEIGHT AT %DB231.DBD1222, 1 s

HMI tags "Data Record DR17"
   "WP231PR_DB_DR17_ANA_OUT_VALUE" : Real = PLC WP231PR_DB.DR17.ANA_OUT_VALUE AT %DB231.DBD1238, 1 s

HMI tags "Data Record DR18"
   "WP231PR_DB_DR18_DEF_DIG_OUT_DQ_0" : Bool = PLC WP231PR_DB.DR18.DEF_DIG_OUT_DQ_0 AT %DB231.DBX1255.0, 1 s
   "WP231PR_DB_DR18_DEF_DIG_OUT_DQ_1" : Bool = PLC WP231PR_DB.DR18.DEF_DIG_OUT_DQ_1 AT %DB231.DBX1255.1, 1 s
   "WP231PR_DB_DR18_DEF_DIG_OUT_DQ_2" : Bool = PLC WP231PR_DB.DR18.DEF_DIG_OUT_DQ_2 AT %DB231.DBX1255.2, 1 s
   "WP231PR_DB_DR18_DEF_DIG_OUT_DQ_3" : Bool = PLC WP231PR_DB.DR18.DEF_DIG_OUT_DQ_3 AT %DB231.DBX1255.3, 1 s

HMI tags "Data Record DR30"
   "WP231PR_DB_DR30_OPERATION_ERRORS" : UInt = PLC WP231PR_DB.DR30.OPERATION_ERRORS AT %DB231.DBW1270, 1 s
   "WP231PR_DB_DR30_TECHNOLOGICAL_ERRORS" : UInt = PLC WP231PR_DB.DR30.TECHNOLOGICAL_ERRORS AT %DB231.DBW1272, 1 s
   "WP231PR_DB_DR30_GROSS_PROCESS" : Real = PLC WP231PR_DB.DR30.GROSS_PROCESS AT %DB231.DBD1274, 500 ms
   "WP231PR_DB_DR30_NET_PROCESS" : Real = PLC WP231PR_DB.DR30.NET_PROCESS AT %DB231.DBD1278, 1 s
   "WP231PR_DB_DR30_TARE_PROCESS" : Real = PLC WP231PR_DB.DR30.TARE_PROCESS AT %DB231.DBD1282, 1 s
   "WP231PR_DB_DR30_GROSS_NET_WEIGHT" : Real = PLC WP231PR_DB.DR30.GROSS_NET_WEIGHT AT %DB231.DBD1286, 1 s
   "WP231PR_DB_DR30_GROSS_NET_WEIGHT_X10" : Real = PLC WP231PR_DB.DR30.GROSS_NET_WEIGHT_X10 AT %DB231.DBD1290, 1 s
   "WP231PR_DB_DR30_TARE" : Real = PLC WP231PR_DB.DR30.TARE AT %DB231.DBD1294, 1 s
   "WP231PR_DB_DR30_GROSS_PROCESS_2" : Real = PLC WP231PR_DB.DR30.GROSS_PROCESS_2 AT %DB231.DBD1298, 1 s
   "WP231PR_DB_DR30_NET_PROCESS_2" : Real = PLC WP231PR_DB.DR30.NET_PROCESS_2 AT %DB231.DBD1302, 1 s
   "WP231PR_DB_DR30_REFRESH_COUNTER" : UInt = PLC WP231PR_DB.DR30.REFRESH_COUNTER AT %DB231.DBW1306, 1 s
   "WP231PR_DB_DR30_LAST_PROTOCOL_ID" : UDInt = PLC WP231PR_DB.DR30.LAST_PROTOCOL_ID AT %DB231.DBD1310, 1 s

HMI tags "Data Record DR31"
   "WP231PR_DB_DR31_DIGITS_UNFILTERED" : DInt = PLC WP231PR_DB.DR31.DIGITS_UNFILTERED AT %DB231.DBD1326, 1 s
   "WP231PR_DB_DR31_DIGITS_FILTERED" : DInt = PLC WP231PR_DB.DR31.DIGITS_FILTERED AT %DB231.DBD1330, 1 s
   "WP231PR_DB_DR31_DIGITS_2_FILTERED" : DInt = PLC WP231PR_DB.DR31.DIGITS_2_FILTERED AT %DB231.DBD1334, 1 s
   "WP231PR_DB_DR31_CURRENT_ANA_OUT_DIGITS" : UInt = PLC WP231PR_DB.DR31.CURRENT_ANA_OUT_DIGITS AT %DB231.DBW1340, 1 s
   "WP231PR_DB_DR31_CURRENT_STATE_DQ_0" : Bool = PLC WP231PR_DB.DR31.CURRENT_STATE_DQ_0 AT %DB231.DBX1342.0, 1 s
   "WP231PR_DB_DR31_CURRENT_STATE_DQ_1" : Bool = PLC WP231PR_DB.DR31.CURRENT_STATE_DQ_1 AT %DB231.DBX1342.1, 1 s
   "WP231PR_DB_DR31_CURRENT_STATE_DQ_2" : Bool = PLC WP231PR_DB.DR31.CURRENT_STATE_DQ_2 AT %DB231.DBX1342.2, 1 s
   "WP231PR_DB_DR31_CURRENT_STATE_DQ_3" : Bool = PLC WP231PR_DB.DR31.CURRENT_STATE_DQ_3 AT %DB231.DBX1342.3, 1 s
   "WP231PR_DB_DR31_CURRENT_STATE_DI_0" : Bool = PLC WP231PR_DB.DR31.CURRENT_STATE_DI_0 AT %DB231.DBX1343.0, 1 s
   "WP231PR_DB_DR31_CURRENT_STATE_DI_1" : Bool = PLC WP231PR_DB.DR31.CURRENT_STATE_DI_1 AT %DB231.DBX1343.1, 1 s
   "WP231PR_DB_DR31_CURRENT_STATE_DI_2" : Bool = PLC WP231PR_DB.DR31.CURRENT_STATE_DI_2 AT %DB231.DBX1343.2, 1 s
   "WP231PR_DB_DR31_CURRENT_STATE_DI_3" : Bool = PLC WP231PR_DB.DR31.CURRENT_STATE_DI_3 AT %DB231.DBX1343.3, 1 s
   "WP231PR_DB_DR31_DIP_SWITCH_1" : Bool = PLC WP231PR_DB.DR31.DIP_SWITCH_1 AT %DB231.DBX1343.6, 1 s
   "WP231PR_DB_DR31_DIP_SWITCH_2" : Bool = PLC WP231PR_DB.DR31.DIP_SWITCH_2 AT %DB231.DBX1343.7, 1 s
   "WP231PR_DB_DR31_REFRESH_COUNTER" : UInt = PLC WP231PR_DB.DR31.REFRESH_COUNTER AT %DB231.DBW1344, 1 s
   "WP231PR_DB_DR31_LOAD_CELL_SIGNAL" : Real = PLC WP231PR_DB.DR31.LOAD_CELL_SIGNAL AT %DB231.DBD1346, 1 s

HMI tags "Data Record DR32"
   "WP231PR_DB_DR32_DATA_CMD_ERR_1" : UInt = PLC WP231PR_DB.DR32.DATA_CMD_ERR_1 AT %DB231.DBW1358, 1 s
   "WP231PR_DB_DR32_DATA_CMD_ERR_2" : UInt = PLC WP231PR_DB.DR32.DATA_CMD_ERR_2 AT %DB231.DBW1360, 1 s
   "WP231PR_DB_DR32_DATA_CMD_ERR_3" : UInt = PLC WP231PR_DB.DR32.DATA_CMD_ERR_3 AT %DB231.DBW1362, 1 s
   "WP231PR_DB_DR32_DATA_CMD_ERR_4" : UInt = PLC WP231PR_DB.DR32.DATA_CMD_ERR_4 AT %DB231.DBW1364, 1 s
   "WP231PR_DB_DR32_ERR_CODE_S7_INTERFACE" : UInt = PLC WP231PR_DB.DR32.ERR_CODE_S7_INTERFACE AT %DB231.DBW1366, 1 s
   "WP231PR_DB_DR32_ERR_CODE_MODBUS_RS485" : UInt = PLC WP231PR_DB.DR32.ERR_CODE_MODBUS_RS485 AT %DB231.DBW1368, 1 s
   "WP231PR_DB_DR32_ERR_CODE_MODBUS_ETH" : UInt = PLC WP231PR_DB.DR32.ERR_CODE_MODBUS_ETH AT %DB231.DBW1370, 1 s
   "WP231PR_DB_DR32_ERR_CODE_SIWATOOL" : UInt = PLC WP231PR_DB.DR32.ERR_CODE_SIWATOOL AT %DB231.DBW1372, 1 s
   "WP231PR_DB_DR32_CMD_ERR_DI" : UInt = PLC WP231PR_DB.DR32.CMD_ERR_DI AT %DB231.DBW1374, 1 s

HMI tags "Data Record DR34"
   "WP231PR_DB_DR34_ASCII_DISPLAY" : String[16] = PLC WP231PR_DB.DR34.ASCII_DISPLAY AT %DB231.DBX1386.0, 100 ms

HMI tags "Data Record DR45"
   "WP231PR_DB_DR45_PROTOCOL_ID_TO_READ" : String[12] = PLC WP231PR_DB.DR45.PROTOCOL_ID_TO_READ AT %DB231.DBX1596.0, 1 s
   "WP231PR_DB_DR45_PROTOCOL_ID_TO_READ_DEC" : DInt = PLC WP231PR_DB.DR45.PROTOCOL_ID_TO_READ_DEC AT %DB231.DBD1612, 1 s

HMI tags "Data Record DR46"
   "WP231PR_DB_DR46_OLDEST_LOG_ID_DEC" : UDInt = PLC WP231PR_DB.DR46.OLDEST_LOG_ID_DEC AT %DB231.DBD1624, 1 s
   "WP231PR_DB_DR46_LAST_LOG_ID_DEC" : UDInt = PLC WP231PR_DB.DR46.LAST_LOG_ID_DEC AT %DB231.DBD1628, 1 s
   "WP231PR_DB_DR46_SELECTED_PROTOCOL_ID_DEC" : UDInt = PLC WP231PR_DB.DR46.SELECTED_PROTOCOL_ID_DEC AT %DB231.DBD1632, 1 s
   "WP231PR_DB_DR46_OLDEST_LOG_ID" : String[12] = PLC WP231PR_DB.DR46.OLDEST_LOG_ID AT %DB231.DBX1636.0, 1 s
   "WP231PR_DB_DR46_LAST_LOG_ID" : String[12] = PLC WP231PR_DB.DR46.LAST_LOG_ID AT %DB231.DBX1650.0, 1 s
   "WP231PR_DB_DR46_SELECTED_PROTOCOL_ID" : String[12] = PLC WP231PR_DB.DR46.SELECTED_PROTOCOL_ID AT %DB231.DBX1664.0, 1 s
   "WP231PR_DB_DR46_PROTOCOL_STRING" : String[28] = PLC WP231PR_DB.DR46.PROTOCOL_STRING AT %DB231.DBX1678.0, 1 s
   "WP231PR_DB_DR46_CHECKSUM" : String[4] = PLC WP231PR_DB.DR46.CHECKSUM AT %DB231.DBX1708.0, 1 s
   "WP231PR_DB_DR46_PROTOCOL_DATE" : String[10] = PLC WP231PR_DB.DR46.PROTOCOL_DATE AT %DB231.DBX1714.0, 1 s
   "WP231PR_DB_DR46_PROTOCOL_TIME" : String[8] = PLC WP231PR_DB.DR46.PROTOCOL_TIME AT %DB231.DBX1726.0, 1 s
   "WP231PR_DB_DR46_ADD_INFORMATION" : String[4] = PLC WP231PR_DB.DR46.ADD_INFORMATION AT %DB231.DBX1736.0, 1 s

HMI tags "Data Record DR47"
   "WP231PR_DB_DR47_OLDEST_LOG_ID" : String[8] = PLC WP231PR_DB.DR47.OLDEST_LOG_ID AT %DB231.DBX1752.0, 1 s
   "WP231PR_DB_DR47_LAST_LOG_ID" : String[8] = PLC WP231PR_DB.DR47.LAST_LOG_ID AT %DB231.DBX1762.0, 1 s
   "WP231PR_DB_DR47_SELECTED_LOG" : String[8] = PLC WP231PR_DB.DR47.SELECTED_LOG AT %DB231.DBX1772.0, 1 s
   "WP231PR_DB_DR47_DEVICE" : String[4] = PLC WP231PR_DB.DR47.DEVICE AT %DB231.DBX1782.0, 1 s
   "WP231PR_DB_DR47_FW_VERSION_OLD" : String[10] = PLC WP231PR_DB.DR47.FW_VERSION_OLD AT %DB231.DBX1788.0, 1 s
   "WP231PR_DB_DR47_FW_VERSION_NEW" : String[10] = PLC WP231PR_DB.DR47.FW_VERSION_NEW AT %DB231.DBX1800.0, 1 s
   "WP231PR_DB_DR47_CHECKSUM" : UInt = PLC WP231PR_DB.DR47.CHECKSUM AT %DB231.DBW1812, 1 s

HMI tags "Data Record DR48"
   "WP231PR_DB_DR48_YEAR" : UInt = PLC WP231PR_DB.DR48.YEAR AT %DB231.DBW1824, 1 s
   "WP231PR_DB_DR48_MONTH" : UInt = PLC WP231PR_DB.DR48.MONTH AT %DB231.DBW1826, 1 s
   "WP231PR_DB_DR48_DAY" : UInt = PLC WP231PR_DB.DR48.DAY AT %DB231.DBW1828, 1 s
   "WP231PR_DB_DR48_HOUR" : UInt = PLC WP231PR_DB.DR48.HOUR AT %DB231.DBW1830, 1 s
   "WP231PR_DB_DR48_MINUTE" : UInt = PLC WP231PR_DB.DR48.MINUTE AT %DB231.DBW1832, 1 s
   "WP231PR_DB_DR48_SECOND" : UInt = PLC WP231PR_DB.DR48.SECOND AT %DB231.DBW1834, 1 s
   "WP231PR_DB_DR48_MSECOND" : UInt = PLC WP231PR_DB.DR48.MSECOND AT %DB231.DBW1836, 1 s
   "WP231PR_DB_DR48_DAY_OF_WEEK" : UInt = PLC WP231PR_DB.DR48.DAY_OF_WEEK AT %DB231.DBW1838, 1 s

HMI tags "CMD"
   "WP231PR_DB_s_CMD1_i_CMD_CODE" : Int = PLC WP231PR_DB.s_CMD1.i_CMD_CODE AT %DB231.DBW462, 1 s
   "WP231PR_DB_s_CMD1_bo_CMD_TRIGGER" : Bool = PLC WP231PR_DB.s_CMD1.bo_CMD_TRIGGER AT %DB231.DBX464.0, 1 s
   "WP231PR_DB_s_CMD2_i_CMD_CODE" : Int = PLC WP231PR_DB.s_CMD2.i_CMD_CODE AT %DB231.DBW466, 1 s
   "WP231PR_DB_s_CMD2_bo_CMD_TRIGGER" : Bool = PLC WP231PR_DB.s_CMD2.bo_CMD_TRIGGER AT %DB231.DBX468.0, 1 s
   "WP231PR_DB_s_CMD3_i_CMD_CODE" : Int = PLC WP231PR_DB.s_CMD3.i_CMD_CODE AT %DB231.DBW470, 1 s
   "WP231PR_DB_s_CMD3_bo_CMD_TRIGGER" : Bool = PLC WP231PR_DB.s_CMD3.bo_CMD_TRIGGER AT %DB231.DBX472.0, 1 s
   "WP231PR_DB_CMD_A" : Int = PLC WP231PR_DB.CMD_A AT %DB231.DBW458, 1 s
   "WP231PR_DB_CMD_B" : Int = PLC WP231PR_DB.CMD_B AT %DB231.DBW460, 1 s

HMI tags "IO_Data"
   "WP231PR_DB_s_IO_DATA_OPERATION_ERRORS" : UInt = PLC WP231PR_DB.s_IO_DATA.OPERATION_ERRORS AT %DB231.DBW508, 100 ms
   "WP231PR_DB_s_IO_DATA_TECHNOLOGICAL_ERRORS" : UInt = PLC WP231PR_DB.s_IO_DATA.TECHNOLOGICAL_ERRORS AT %DB231.DBW510, 100 ms
   "WP231PR_DB_s_IO_DATA_DATA_CMD_ERROR_1" : UInt = PLC WP231PR_DB.s_IO_DATA.DATA_CMD_ERROR_1 AT %DB231.DBW512, 100 ms
   "WP231PR_DB_s_IO_DATA_DATA_CMD_ERROR_2" : UInt = PLC WP231PR_DB.s_IO_DATA.DATA_CMD_ERROR_2 AT %DB231.DBW514, 100 ms
   "WP231PR_DB_s_IO_DATA_DATA_CMD_ERROR_3" : UInt = PLC WP231PR_DB.s_IO_DATA.DATA_CMD_ERROR_3 AT %DB231.DBW516, 100 ms
   "WP231PR_DB_s_IO_DATA_DATA_CMD_ERROR_4" : UInt = PLC WP231PR_DB.s_IO_DATA.DATA_CMD_ERROR_4 AT %DB231.DBW518, 100 ms
   "WP231PR_DB_s_IO_DATA_SCALE_STATUS_1_EMPTY" : Bool = PLC WP231PR_DB.s_IO_DATA.SCALE_STATUS_1.EMPTY AT %DB231.DBX488.0, 100 ms
   "WP231PR_DB_s_IO_DATA_SCALE_STATUS_1_LIMIT_1" : Bool = PLC WP231PR_DB.s_IO_DATA.SCALE_STATUS_1.LIMIT_1 AT %DB231.DBX488.1, 100 ms
   "WP231PR_DB_s_IO_DATA_SCALE_STATUS_1_LIMIT_2" : Bool = PLC WP231PR_DB.s_IO_DATA.SCALE_STATUS_1.LIMIT_2 AT %DB231.DBX488.2, 100 ms
   "WP231PR_DB_s_IO_DATA_SCALE_STATUS_1_BELOW_MIN_WEIGHT" : Bool = PLC WP231PR_DB.s_IO_DATA.SCALE_STATUS_1.BELOW_MIN_WEIGHT AT %DB231.DBX488.3, 100 ms
   "WP231PR_DB_s_IO_DATA_SCALE_STATUS_1_D_ZERO" : Bool = PLC WP231PR_DB.s_IO_DATA.SCALE_STATUS_1.D_ZERO AT %DB231.DBX489.0, 100 ms
   "WP231PR_DB_s_IO_DATA_SCALE_STATUS_1_MAX_9E" : Bool = PLC WP231PR_DB.s_IO_DATA.SCALE_STATUS_1.MAX_9E AT %DB231.DBX489.1, 100 ms
   "WP231PR_DB_s_IO_DATA_SCALE_STATUS_1_TARE" : Bool = PLC WP231PR_DB.s_IO_DATA.SCALE_STATUS_1.TARE AT %DB231.DBX489.2, 100 ms
   "WP231PR_DB_s_IO_DATA_SCALE_STATUS_1_PRESET_TARE" : Bool = PLC WP231PR_DB.s_IO_DATA.SCALE_STATUS_1.PRESET_TARE AT %DB231.DBX489.3, 100 ms
   "WP231PR_DB_s_IO_DATA_SCALE_STATUS_1_WAITING_FOR_STANDSTILL" : Bool = PLC WP231PR_DB.s_IO_DATA.SCALE_STATUS_1.WAITING_FOR_STANDSTILL AT %DB231.DBX489.5, 100 ms
   "WP231PR_DB_s_IO_DATA_SCALE_STATUS_1_STANDSTILL" : Bool = PLC WP231PR_DB.s_IO_DATA.SCALE_STATUS_1.STANDSTILL AT %DB231.DBX489.6, 100 ms
   "WP231PR_DB_s_IO_DATA_SCALE_STATUS_2_CALIBRATED" : Bool = PLC WP231PR_DB.s_IO_DATA.SCALE_STATUS_2.CALIBRATED AT %DB231.DBX490.0, 100 ms
   "WP231PR_DB_s_IO_DATA_SCALE_STATUS_2_SERVICE_MODE" : Bool = PLC WP231PR_DB.s_IO_DATA.SCALE_STATUS_2.SERVICE_MODE AT %DB231.DBX490.1, 100 ms
   "WP231PR_DB_s_IO_DATA_SCALE_STATUS_2_SIMULATION_MODE" : Bool = PLC WP231PR_DB.s_IO_DATA.SCALE_STATUS_2.SIMULATION_MODE AT %DB231.DBX490.2, 100 ms
   "WP231PR_DB_s_IO_DATA_SCALE_STATUS_2_WRITE_PROTECTION" : Bool = PLC WP231PR_DB.s_IO_DATA.SCALE_STATUS_2.WRITE_PROTECTION AT %DB231.DBX490.3, 100 ms
   "WP231PR_DB_s_IO_DATA_SCALE_STATUS_2_ANALOGUE_OUT_ERROR" : Bool = PLC WP231PR_DB.s_IO_DATA.SCALE_STATUS_2.ANALOGUE_OUT_ERROR AT %DB231.DBX490.4, 100 ms
   "WP231PR_DB_s_IO_DATA_SCALE_STATUS_2_START_UP" : Bool = PLC WP231PR_DB.s_IO_DATA.SCALE_STATUS_2.START_UP AT %DB231.DBX490.6, 100 ms
   "WP231PR_DB_s_IO_DATA_SCALE_STATUS_2_ERROR" : Bool = PLC WP231PR_DB.s_IO_DATA.SCALE_STATUS_2.ERROR AT %DB231.DBX490.7, 100 ms
   "WP231PR_DB_s_IO_DATA_SCALE_STATUS_2_TIME_BUFFER_ERROR" : Bool = PLC WP231PR_DB.s_IO_DATA.SCALE_STATUS_2.TIME_BUFFER_ERROR AT %DB231.DBX491.5, 100 ms
   "WP231PR_DB_s_IO_DATA_SCALE_STATUS_2_TRACE" : Bool = PLC WP231PR_DB.s_IO_DATA.SCALE_STATUS_2.TRACE AT %DB231.DBX491.6, 100 ms
   "WP231PR_DB_s_IO_DATA_SCALE_STATUS_2_DIGITAL_INPUT_ERROR" : Bool = PLC WP231PR_DB.s_IO_DATA.SCALE_STATUS_2.DIGITAL_INPUT_ERROR AT %DB231.DBX491.7, 100 ms

HMI tags "INTERNAL"
   "S1_DISPLAY_TAG" : Bool, internal
   "S1_LOADCURVE_MIN" : Real, internal
   "S1_SHOW_HELP" : Bool, internal
   "SecureDisplayRunning" : Bool AT %DB1.DBX0.0

